LIN {X 0,Y 311.55,Z 599.519,A -85,B 0,C 180,E1 -15563.524,E2 -15563.524} C_VEL
LIN {X 0,Y 311.702,Z 601.489,A -85,B 0,C 180,E1 -15564.826,E2 -15564.826} C_VEL
LIN {X 0,Y 311.941,Z 602.986,A -85,B 0,C 180,E1 -15566.124,E2 -15566.124} C_VEL
LIN {X 0,Y 312.344,Z 604.721,A -85,B 0,C 180,E1 -15568.711,E2 -15568.711} C_VEL
LIN {X 0,Y 312.557,Z 604.974,A -85,B 0,C 180,E1 -15570,E2 -15570} C_VEL
LIN {X 0,Y 312.346,Z 604.715,A -85,B 0,C 180,E1 -15571.289,E2 -15571.289} C_VEL
LIN {X 0,Y 311.948,Z 602.974,A -85,B 0,C 180,E1 -15573.875,E2 -15573.875} C_VEL
LIN {X 0,Y 311.715,Z 601.472,A -85,B 0,C 180,E1 -15575.174,E2 -15575.174} C_VEL
LIN {X 0,Y 311.515,Z 598.688,A -85,B 0,C 180,E1 -15576.94,E2 -15576.94} C_VEL
LIN {X 0,Y 311.364,Z 594.173,A -85,B 0,C 180,E1 -15579.091,E2 -15579.091} C_VEL
LIN {X 0,Y 311.678,Z 587.813,A -85,B 0,C 180,E1 -15581.379,E2 -15581.379} C_VEL
LIN {X 0,Y 312.28,Z 580.919,A -85,B 0,C 180,E1 -15583.337,E2 -15583.337} C_VEL
LIN {X 0,Y 313.101,Z 573.765,A -85,B 0,C 180,E1 -15584.999,E2 -15584.999} C_VEL
LIN {X 0,Y 314.326,Z 565.613,A -85,B 0,C 180,E1 -15586.563,E2 -15586.563} C_VEL
LIN {X 0,Y 315.624,Z 556.565,A -85,B 0,C 180,E1 -15587.996,E2 -15587.996} C_VEL
LIN {X 0,Y 317.241,Z 545.513,A -85,B 0,C 180,E1 -15589.408,E2 -15589.408} C_VEL
LIN {X 0,Y 318.954,Z 532.942,A -85,B 0,C 180,E1 -15590.643,E2 -15590.643} C_VEL
LIN {X 0,Y 320.384,Z 520.621,A -85,B 0,C 180,E1 -15591.557,E2 -15591.557} C_VEL
LIN {X 0,Y 321.477,Z 507.646,A -85,B 0,C 180,E1 -15592.239,E2 -15592.239} C_VEL
LIN {X 0,Y 322.122,Z 493.846,A -85,B 0,C 180,E1 -15592.699,E2 -15592.699} C_VEL
LIN {X 0,Y 323.046,Z 447.747,A -85,B 0,C 180,E1 -15593.723,E2 -15593.723} C_VEL
LIN {X 0,Y 319.721,Z 414.393,A -85,B 0,C 180,E1 -15594.772,E2 -15594.772} C_VEL
LIN {X 0,Y 316.416,Z 387.78,A -85,B 0,C 180,E1 -15595.724,E2 -15595.724} C_VEL
LIN {X 0,Y 319.076,Z 366.674,A -85,B 0,C 180,E1 -15600.072,E2 -15600.072} C_VEL
LIN {X 0,Y 319.477,Z 362.665,A -85,B 0,C 180,E1 -15600.914,E2 -15600.914} C_VEL
LIN {X 0,Y 317.162,Z 351.199,A -85,B 0,C 180,E1 -15603.639,E2 -15603.639} C_VEL
LIN {X 0,Y 314.169,Z 338.968,A -85,B 0,C 180,E1 -15606.716,E2 -15606.716} C_VEL
LIN {X 0,Y 312.497,Z 332.686,A -85,B 0,C 180,E1 -15608.434,E2 -15608.434} C_VEL
LIN {X 0,Y 312.462,Z 332.564,A -85,B 0,C 180,E1 -15612.435,E2 -15612.435} C_VEL
LIN {X 0,Y 312.452,Z 332.533,A -85,B 0,C 180,E1 -15616.035,E2 -15616.035} C_VEL
LIN {X 0,Y 312.451,Z 332.552,A -85,B 0,C 180,E1 -15619.885,E2 -15619.885} C_VEL
LIN {X 0,Y 312.528,Z 332.497,A -85,B 0,C 180,E1 -15624.051,E2 -15624.051} C_VEL
LIN {X 0,Y 312.497,Z 332.555,A -85,B 0,C 180,E1 -15627.333,E2 -15627.333} C_VEL
LIN {X 0,Y 312.501,Z 332.536,A -85,B 0,C 180,E1 -15631.291,E2 -15631.291} C_VEL
LIN {X 0,Y 312.52,Z 332.555,A -85,B 0,C 180,E1 -15634.705,E2 -15634.705} C_VEL
LIN {X 0,Y 312.529,Z 332.523,A -85,B 0,C 180,E1 -15638.912,E2 -15638.912} C_VEL
LIN {X 0,Y 312.633,Z 332.53,A -85,B 0,C 180,E1 -15641.656,E2 -15641.656} C_VEL
LIN {X 0,Y 312.688,Z 332.525,A -85,B 0,C 180,E1 -15645.686,E2 -15645.686} C_VEL
LIN {X 0,Y 312.679,Z 332.535,A -85,B 0,C 180,E1 -15649.641,E2 -15649.641} C_VEL
LIN {X 0,Y 312.813,Z 332.51,A -85,B 0,C 180,E1 -15652.253,E2 -15652.253} C_VEL
LIN {X 0,Y 312.686,Z 332.523,A -85,B 0,C 180,E1 -15654.842,E2 -15654.842} C_VEL
LIN {X 0,Y 312.973,Z 332.495,A -85,B 0,C 180,E1 -15658.713,E2 -15658.713} C_VEL
LIN {X 0,Y 312.902,Z 332.502,A -85,B 0,C 180,E1 -15662.575,E2 -15662.575} C_VEL
LIN {X 0,Y 312.831,Z 332.506,A -85,B 0,C 180,E1 -15666.473,E2 -15666.473} C_VEL
LIN {X 0,Y 312.745,Z 332.515,A -85,B 0,C 180,E1 -15669.051,E2 -15669.051} C_VEL
LIN {X 0,Y 312.627,Z 332.536,A -85,B 0,C 180,E1 -15672.991,E2 -15672.991} C_VEL
LIN {X 0,Y 312.616,Z 332.531,A -85,B 0,C 180,E1 -15675.651,E2 -15675.651} C_VEL
LIN {X 0,Y 312.554,Z 332.542,A -85,B 0,C 180,E1 -15679.712,E2 -15679.712} C_VEL
LIN {X 0,Y 312.509,Z 332.553,A -85,B 0,C 180,E1 -15682.775,E2 -15682.775} C_VEL
LIN {X 0,Y 312.477,Z 332.543,A -85,B 0,C 180,E1 -15686.733,E2 -15686.733} C_VEL
LIN {X 0,Y 312.462,Z 332.51,A -85,B 0,C 180,E1 -15689.659,E2 -15689.659} C_VEL
LIN {X 0,Y 312.516,Z 332.553,A -85,B 0,C 180,E1 -15693.689,E2 -15693.689} C_VEL
LIN {X 0,Y 312.506,Z 332.535,A -85,B 0,C 180,E1 -15697.388,E2 -15697.388} C_VEL
LIN {X 0,Y 312.437,Z 332.541,A -85,B 0,C 180,E1 -15700.718,E2 -15700.718} C_VEL
LIN {X 0,Y 312.447,Z 332.562,A -85,B 0,C 180,E1 -15704.211,E2 -15704.211} C_VEL
LIN {X 0,Y 312.451,Z 332.544,A -85,B 0,C 180,E1 -15707.926,E2 -15707.926} C_VEL
LIN {X 0,Y 312.481,Z 332.544,A -85,B 0,C 180,E1 -15711.923,E2 -15711.923} C_VEL
LIN {X 0,Y 312.528,Z 332.548,A -85,B 0,C 180,E1 -15714.221,E2 -15714.221} C_VEL
LIN {X 0,Y 312.5,Z 332.545,A -85,B 0,C 180,E1 -15717.334,E2 -15717.334} C_VEL
LIN {X 0,Y 312.483,Z 332.528,A -85,B 0,C 180,E1 -15721.3,E2 -15721.3} C_VEL
LIN {X 0,Y 312.579,Z 332.675,A -85,B 0,C 180,E1 -15724.399,E2 -15724.399} C_VEL
LIN {X 0,Y 312.787,Z 333.571,A -85,B 0,C 180,E1 -15724.634,E2 -15724.634} C_VEL
LIN {X 0,Y 322.25,Z 353.976,A -85,B 0,C 180,E1 -15725.982,E2 -15725.982} C_VEL
LIN {X 0,Y 324.863,Z 359.97,A -85,B 0,C 180,E1 -15726.34,E2 -15726.34} C_VEL
LIN {X 0,Y 324.035,Z 414.568,A -85,B 0,C 180,E1 -15727.593,E2 -15727.593} C_VEL
LIN {X 0,Y 323.772,Z 427.043,A -85,B 0,C 180,E1 -15728.1,E2 -15728.1} C_VEL
LIN {X 0,Y 323.165,Z 439.993,A -85,B 0,C 180,E1 -15728.889,E2 -15728.889} C_VEL
LIN {X 0,Y 322.296,Z 452.305,A -85,B 0,C 180,E1 -15729.911,E2 -15729.911} C_VEL
LIN {X 0,Y 320.98,Z 463.869,A -85,B 0,C 180,E1 -15731.159,E2 -15731.159} C_VEL
LIN {X 0,Y 319.694,Z 474.198,A -85,B 0,C 180,E1 -15732.571,E2 -15732.571} C_VEL
LIN {X 0,Y 318.595,Z 482.613,A -85,B 0,C 180,E1 -15733.994,E2 -15733.994} C_VEL
LIN {X 0,Y 317.424,Z 490.361,A -85,B 0,C 180,E1 -15735.577,E2 -15735.577} C_VEL
LIN {X 0,Y 316.218,Z 498.029,A -85,B 0,C 180,E1 -15737.518,E2 -15737.518} C_VEL
LIN {X 0,Y 315.27,Z 503.78,A -85,B 0,C 180,E1 -15739.336,E2 -15739.336} C_VEL
LIN {X 0,Y 314.62,Z 508.048,A -85,B 0,C 180,E1 -15741.004,E2 -15741.004} C_VEL
LIN {X 0,Y 313.789,Z 511.941,A -85,B 0,C 180,E1 -15742.924,E2 -15742.924} C_VEL
LIN {X 0,Y 313.156,Z 514.815,A -85,B 0,C 180,E1 -15744.85,E2 -15744.85} C_VEL
LIN {X 0,Y 313.098,Z 516.157,A -85,B 0,C 180,E1 -15746.139,E2 -15746.139} C_VEL
LIN {X 0,Y 312.876,Z 517.135,A -85,B 0,C 180,E1 -15747.425,E2 -15747.425} C_VEL
LIN {X 0,Y 312.907,Z 517.715,A -85,B 0,C 180,E1 -15748.713,E2 -15748.713} C_VEL
LIN {X 0,Y 312.881,Z 517.941,A -85,B 0,C 180,E1 -15750,E2 -15750} C_VEL
LIN {X 0,Y 312.907,Z 517.755,A -85,B 0,C 180,E1 -15751.287,E2 -15751.287} C_VEL
LIN {X 0,Y 312.875,Z 517.201,A -85,B 0,C 180,E1 -15752.575,E2 -15752.575} C_VEL
LIN {X 0,Y 313.093,Z 516.248,A -85,B 0,C 180,E1 -15753.861,E2 -15753.861} C_VEL
LIN {X 0,Y 313.144,Z 514.948,A -85,B 0,C 180,E1 -15755.15,E2 -15755.15} C_VEL
LIN {X 0,Y 313.783,Z 512.122,A -85,B 0,C 180,E1 -15757.076,E2 -15757.076} C_VEL
LIN {X 0,Y 314.595,Z 508.294,A -85,B 0,C 180,E1 -15758.997,E2 -15758.997} C_VEL
LIN {X 0,Y 315.35,Z 503.213,A -85,B 0,C 180,E1 -15760.984,E2 -15760.984} C_VEL
LIN {X 0,Y 316.648,Z 495.971,A -85,B 0,C 180,E1 -15763.15,E2 -15763.15} C_VEL
LIN {X 0,Y 317.934,Z 487.942,A -85,B 0,C 180,E1 -15765.054,E2 -15765.054} C_VEL
LIN {X 0,Y 319.058,Z 479.718,A -85,B 0,C 180,E1 -15766.64,E2 -15766.64} C_VEL
LIN {X 0,Y 320.218,Z 470.679,A -85,B 0,C 180,E1 -15768.059,E2 -15768.059} C_VEL
LIN {X 0,Y 321.556,Z 460.163,A -85,B 0,C 180,E1 -15769.378,E2 -15769.378} C_VEL
LIN {X 0,Y 322.613,Z 448.643,A -85,B 0,C 180,E1 -15770.533,E2 -15770.533} C_VEL
LIN {X 0,Y 323.495,Z 437.366,A -85,B 0,C 180,E1 -15771.398,E2 -15771.398} C_VEL
LIN {X 0,Y 323.977,Z 425.075,A -85,B 0,C 180,E1 -15772.098,E2 -15772.098} C_VEL
LIN {X 0,Y 324.096,Z 414.763,A -85,B 0,C 180,E1 -15772.511,E2 -15772.511} C_VEL
LIN {X 0,Y 324.643,Z 374.354,A -85,B 0,C 180,E1 -15773.45,E2 -15773.45} C_VEL
LIN {X 0,Y 324.833,Z 359.99,A -85,B 0,C 180,E1 -15773.776,E2 -15773.776} C_VEL
LIN {X 0,Y 316.003,Z 340.297,A -85,B 0,C 180,E1 -15775.003,E2 -15775.003} C_VEL
LIN {X 0,Y 312.728,Z 333.371,A -85,B 0,C 180,E1 -15775.513,E2 -15775.513} C_VEL
LIN {X 0,Y 312.548,Z 332.615,A -85,B 0,C 180,E1 -15775.775,E2 -15775.775} C_VEL
LIN {X 0,Y 312.467,Z 332.547,A -85,B 0,C 180,E1 -15779.657,E2 -15779.657} C_VEL
LIN {X 0,Y 312.519,Z 332.549,A -85,B 0,C 180,E1 -15783.688,E2 -15783.688} C_VEL
LIN {X 0,Y 312.508,Z 332.537,A -85,B 0,C 180,E1 -15787.387,E2 -15787.387} C_VEL
LIN {X 0,Y 312.438,Z 332.564,A -85,B 0,C 180,E1 -15790.716,E2 -15790.716} C_VEL
LIN {X 0,Y 312.447,Z 332.543,A -85,B 0,C 180,E1 -15794.209,E2 -15794.209} C_VEL
LIN {X 0,Y 312.451,Z 332.562,A -85,B 0,C 180,E1 -15797.924,E2 -15797.924} C_VEL
LIN {X 0,Y 312.422,Z 332.551,A -85,B 0,C 180,E1 -15798.789,E2 -15798.789} C_VEL
LIN {X 0,Y 311.768,Z 332.623,A -85,B 0,C 180,E1 -15799.864,E2 -15799.864} C_VEL
LIN {X 0,Y 308.931,Z 332.977,A -85,B 0,C 180,E1 -15801.614,E2 -15801.614} C_VEL
LIN {X 0,Y 306.53,Z 333.286,A -85,B 0,C 180,E1 -15803.034,E2 -15803.034} C_VEL
LIN {X 0,Y 305.516,Z 333.423,A -85,B 0,C 180,E1 -15804.133,E2 -15804.133} C_VEL
LIN {X 0,Y 305.443,Z 333.435,A -85,B 0,C 180,E1 -15804.505,E2 -15804.505} C_VEL
LIN {X 0,Y 305.437,Z 333.407,A -85,B 0,C 180,E1 -15808.358,E2 -15808.358} C_VEL
LIN {X 0,Y 305.447,Z 333.385,A -85,B 0,C 180,E1 -15811.106,E2 -15811.106} C_VEL
LIN {X 0,Y 305.473,Z 333.423,A -85,B 0,C 180,E1 -15814.079,E2 -15814.079} C_VEL
LIN {X 0,Y 305.455,Z 333.423,A -85,B 0,C 180,E1 -15818.399,E2 -15818.399} C_VEL
LIN {X 0,Y 305.529,Z 333.427,A -85,B 0,C 180,E1 -15822.6,E2 -15822.6} C_VEL
LIN {X 0,Y 305.62,Z 333.395,A -85,B 0,C 180,E1 -15825.347,E2 -15825.347} C_VEL
LIN {X 0,Y 305.618,Z 333.413,A -85,B 0,C 180,E1 -15829.399,E2 -15829.399} C_VEL
LIN {X 0,Y 305.739,Z 333.383,A -85,B 0,C 180,E1 -15832.072,E2 -15832.072} C_VEL
LIN {X 0,Y 305.653,Z 333.412,A -85,B 0,C 180,E1 -15834.723,E2 -15834.723} C_VEL
LIN {X 0,Y 305.929,Z 333.358,A -85,B 0,C 180,E1 -15838.684,E2 -15838.684} C_VEL
LIN {X 0,Y 305.94,Z 333.371,A -85,B 0,C 180,E1 -15841.316,E2 -15841.316} C_VEL
LIN {X 0,Y 305.786,Z 333.378,A -85,B 0,C 180,E1 -15846.599,E2 -15846.599} C_VEL
LIN {X 0,Y 305.688,Z 333.405,A -85,B 0,C 180,E1 -15849.261,E2 -15849.261} C_VEL
LIN {X 0,Y 305.579,Z 333.404,A -85,B 0,C 180,E1 -15853.296,E2 -15853.296} C_VEL
LIN {X 0,Y 305.55,Z 333.425,A -85,B 0,C 180,E1 -15856.022,E2 -15856.022} C_VEL
LIN {X 0,Y 305.537,Z 333.401,A -85,B 0,C 180,E1 -15859.426,E2 -15859.426} C_VEL
LIN {X 0,Y 305.466,Z 333.427,A -85,B 0,C 180,E1 -15863.033,E2 -15863.033} C_VEL
LIN {X 0,Y 305.449,Z 333.43,A -85,B 0,C 180,E1 -15866.191,E2 -15866.191} C_VEL
LIN {X 0,Y 305.443,Z 333.417,A -85,B 0,C 180,E1 -15869.034,E2 -15869.034} C_VEL
LIN {X 0,Y 305.432,Z 333.442,A -85,B 0,C 180,E1 -15871.954,E2 -15871.954} C_VEL
LIN {X 0,Y 305.457,Z 333.421,A -85,B 0,C 180,E1 -15875.114,E2 -15875.114} C_VEL
LIN {X 0,Y 305.43,Z 333.43,A -85,B 0,C 180,E1 -15878.525,E2 -15878.525} C_VEL
LIN {X 0,Y 305.431,Z 333.432,A -85,B 0,C 180,E1 -15882.582,E2 -15882.582} C_VEL
LIN {X 0,Y 305.417,Z 333.412,A -85,B 0,C 180,E1 -15886.344,E2 -15886.344} C_VEL
LIN {X 0,Y 305.407,Z 333.418,A -85,B 0,C 180,E1 -15889.885,E2 -15889.885} C_VEL
LIN {X 0,Y 305.447,Z 333.618,A -85,B 0,C 180,E1 -15890.998,E2 -15890.998} C_VEL
LIN {X 0,Y 308.846,Z 346.507,A -85,B 0,C 180,E1 -15894.491,E2 -15894.491} C_VEL
LIN {X 0,Y 311.665,Z 358.968,A -85,B 0,C 180,E1 -15897.619,E2 -15897.619} C_VEL
LIN {X 0,Y 312.62,Z 364.164,A -85,B 0,C 180,E1 -15898.865,E2 -15898.865} C_VEL
LIN {X 0,Y 311.106,Z 375.627,A -85,B 0,C 180,E1 -15901.312,E2 -15901.312} C_VEL
LIN {X 0,Y 309.717,Z 386.706,A -85,B 0,C 180,E1 -15903.647,E2 -15903.647} C_VEL
LIN {X 0,Y 313.735,Z 419.226,A -85,B 0,C 180,E1 -15904.839,E2 -15904.839} C_VEL
LIN {X 0,Y 316.571,Z 448.811,A -85,B 0,C 180,E1 -15905.787,E2 -15905.787} C_VEL
LIN {X 0,Y 315.459,Z 497.939,A -85,B 0,C 180,E1 -15906.924,E2 -15906.924} C_VEL
LIN {X 0,Y 314.589,Z 511.17,A -85,B 0,C 180,E1 -15907.464,E2 -15907.464} C_VEL
LIN {X 0,Y 313.434,Z 523.348,A -85,B 0,C 180,E1 -15908.2,E2 -15908.2} C_VEL
LIN {X 0,Y 311.838,Z 535.654,A -85,B 0,C 180,E1 -15909.209,E2 -15909.209} C_VEL
LIN {X 0,Y 310.115,Z 547.326,A -85,B 0,C 180,E1 -15910.472,E2 -15910.472} C_VEL
LIN {X 0,Y 308.48,Z 557.874,A -85,B 0,C 180,E1 -15911.916,E2 -15911.916} C_VEL
LIN {X 0,Y 307.228,Z 566.547,A -85,B 0,C 180,E1 -15913.385,E2 -15913.385} C_VEL
LIN {X 0,Y 305.954,Z 574.893,A -85,B 0,C 180,E1 -15915.099,E2 -15915.099} C_VEL
LIN {X 0,Y 305.068,Z 582.466,A -85,B 0,C 180,E1 -15917.02,E2 -15917.02} C_VEL
LIN {X 0,Y 304.448,Z 589.797,A -85,B 0,C 180,E1 -15919.358,E2 -15919.358} C_VEL
LIN {X 0,Y 304.276,Z 594.719,A -85,B 0,C 180,E1 -15921.365,E2 -15921.365} C_VEL
LIN {X 0,Y 304.443,Z 598.525,A -85,B 0,C 180,E1 -15923.372,E2 -15923.372} C_VEL
LIN {X 0,Y 304.615,Z 600.5,A -85,B 0,C 180,E1 -15924.705,E2 -15924.705} C_VEL
LIN {X 0,Y 304.869,Z 602,A -85,B 0,C 180,E1 -15926.034,E2 -15926.034} C_VEL
LIN {X 0,Y 305.285,Z 603.738,A -85,B 0,C 180,E1 -15928.681,E2 -15928.681} C_VEL
LIN {X 0,Y 305.525,Z 603.995,A -85,B 0,C 180,E1 -15930,E2 -15930} C_VEL
LIN {X 0,Y 305.287,Z 603.732,A -85,B 0,C 180,E1 -15931.319,E2 -15931.319} C_VEL
LIN {X 0,Y 304.894,Z 601.99,A -85,B 0,C 180,E1 -15933.965,E2 -15933.965} C_VEL
LIN {X 0,Y 304.631,Z 600.482,A -85,B 0,C 180,E1 -15935.295,E2 -15935.295} C_VEL
LIN {X 0,Y 304.438,Z 597.963,A -85,B 0,C 180,E1 -15936.944,E2 -15936.944} C_VEL
LIN {X 0,Y 304.31,Z 593.178,A -85,B 0,C 180,E1 -15939.303,E2 -15939.303} C_VEL
LIN {X 0,Y 304.663,Z 586.816,A -85,B 0,C 180,E1 -15941.645,E2 -15941.645} C_VEL
LIN {X 0,Y 305.331,Z 579.923,A -85,B 0,C 180,E1 -15943.646,E2 -15943.646} C_VEL
LIN {X 0,Y 306.333,Z 572.003,A -85,B 0,C 180,E1 -15945.51,E2 -15945.51} C_VEL
LIN {X 0,Y 307.655,Z 562.765,A -85,B 0,C 180,E1 -15947.275,E2 -15947.275} C_VEL
LIN {X 0,Y 309.372,Z 552.132,A -85,B 0,C 180,E1 -15948.887,E2 -15948.887} C_VEL
LIN {X 0,Y 310.967,Z 541.643,A -85,B 0,C 180,E1 -15950.16,E2 -15950.16} C_VEL
LIN {X 0,Y 312.611,Z 530.177,A -85,B 0,C 180,E1 -15951.254,E2 -15951.254} C_VEL
LIN {X 0,Y 313.924,Z 518.382,A -85,B 0,C 180,E1 -15952.11,E2 -15952.11} C_VEL
LIN {X 0,Y 315.03,Z 504.81,A -85,B 0,C 180,E1 -15952.806,E2 -15952.806} C_VEL
LIN {X 0,Y 315.633,Z 491.252,A -85,B 0,C 180,E1 -15953.236,E2 -15953.236} C_VEL
LIN {X 0,Y 316.51,Z 448.386,A -85,B 0,C 180,E1 -15954.204,E2 -15954.204} C_VEL
LIN {X 0,Y 313.251,Z 415.354,A -85,B 0,C 180,E1 -15955.271,E2 -15955.271} C_VEL
LIN {X 0,Y 309.681,Z 387.005,A -85,B 0,C 180,E1 -15956.3,E2 -15956.3} C_VEL
LIN {X 0,Y 310.898,Z 377.146,A -85,B 0,C 180,E1 -15958.34,E2 -15958.34} C_VEL
LIN {X 0,Y 312.586,Z 364.015,A -85,B 0,C 180,E1 -15961.139,E2 -15961.139} C_VEL
LIN {X 0,Y 310.058,Z 351.698,A -85,B 0,C 180,E1 -15964.156,E2 -15964.156} C_VEL
LIN {X 0,Y 307.06,Z 339.565,A -85,B 0,C 180,E1 -15967.309,E2 -15967.309} C_VEL
LIN {X 0,Y 305.436,Z 333.537,A -85,B 0,C 180,E1 -15969.021,E2 -15969.021} C_VEL
LIN {X 0,Y 305.432,Z 333.434,A -85,B 0,C 180,E1 -15972.581,E2 -15972.581} C_VEL
LIN {X 0,Y 305.417,Z 333.413,A -85,B 0,C 180,E1 -15976.343,E2 -15976.343} C_VEL
LIN {X 0,Y 305.406,Z 333.43,A -85,B 0,C 180,E1 -15979.884,E2 -15979.884} C_VEL
LIN {X 0,Y 305.456,Z 333.372,A -85,B 0,C 180,E1 -15983.637,E2 -15983.637} C_VEL
LIN {X 0,Y 305.46,Z 333.423,A -85,B 0,C 180,E1 -15986.483,E2 -15986.483} C_VEL
LIN {X 0,Y 305.426,Z 333.432,A -85,B 0,C 180,E1 -15989.587,E2 -15989.587} C_VEL
LIN {X 0,Y 305.447,Z 333.42,A -85,B 0,C 180,E1 -15992.601,E2 -15992.601} C_VEL
LIN {X 0,Y 305.454,Z 333.438,A -85,B 0,C 180,E1 -15995.534,E2 -15995.534} C_VEL
LIN {X 0,Y 305.5,Z 333.398,A -85,B 0,C 180,E1 -15999.814,E2 -15999.814} C_VEL
LIN {X 0,Y 305.569,Z 333.419,A -85,B 0,C 180,E1 -16002.603,E2 -16002.603} C_VEL
LIN {X 0,Y 305.644,Z 333.407,A -85,B 0,C 180,E1 -16005.349,E2 -16005.349} C_VEL
LIN {X 0,Y 305.618,Z 333.412,A -85,B 0,C 180,E1 -16009.399,E2 -16009.399} C_VEL
LIN {X 0,Y 305.759,Z 333.39,A -85,B 0,C 180,E1 -16012.073,E2 -16012.073} C_VEL
LIN {X 0,Y 305.656,Z 333.398,A -85,B 0,C 180,E1 -16014.723,E2 -16014.723} C_VEL
LIN {X 0,Y 305.94,Z 333.371,A -85,B 0,C 180,E1 -16018.684,E2 -16018.684} C_VEL
LIN {X 0,Y 305.929,Z 333.357,A -85,B 0,C 180,E1 -16021.316,E2 -16021.316} C_VEL
LIN {X 0,Y 305.655,Z 333.411,A -85,B 0,C 180,E1 -16025.277,E2 -16025.277} C_VEL
LIN {X 0,Y 305.739,Z 333.382,A -85,B 0,C 180,E1 -16027.928,E2 -16027.928} C_VEL
LIN {X 0,Y 305.592,Z 333.415,A -85,B 0,C 180,E1 -16031.946,E2 -16031.946} C_VEL
LIN {X 0,Y 305.603,Z 333.398,A -85,B 0,C 180,E1 -16035.014,E2 -16035.014} C_VEL
LIN {X 0,Y 305.537,Z 333.419,A -85,B 0,C 180,E1 -16039.427,E2 -16039.427} C_VEL
LIN {X 0,Y 305.451,Z 333.433,A -85,B 0,C 180,E1 -16043.026,E2 -16043.026} C_VEL
LIN {X 0,Y 305.446,Z 333.425,A -85,B 0,C 180,E1 -16046.19,E2 -16046.19} C_VEL
LIN {X 0,Y 305.418,Z 333.388,A -85,B 0,C 180,E1 -16049.026,E2 -16049.026} C_VEL
LIN {X 0,Y 305.432,Z 333.412,A -85,B 0,C 180,E1 -16051.954,E2 -16051.954} C_VEL
LIN {X 0,Y 305.458,Z 333.437,A -85,B 0,C 180,E1 -16055.114,E2 -16055.114} C_VEL
LIN {X 0,Y 305.43,Z 333.402,A -85,B 0,C 180,E1 -16058.525,E2 -16058.525} C_VEL
LIN {X 0,Y 305.431,Z 333.437,A -85,B 0,C 180,E1 -16062.582,E2 -16062.582} C_VEL
LIN {X 0,Y 305.417,Z 333.413,A -85,B 0,C 180,E1 -16066.345,E2 -16066.345} C_VEL
LIN {X 0,Y 305.408,Z 333.443,A -85,B 0,C 180,E1 -16069.885,E2 -16069.885} C_VEL
LIN {X 0,Y 305.461,Z 333.419,A -85,B 0,C 180,E1 -16073.637,E2 -16073.637} C_VEL
LIN {X 0,Y 305.464,Z 333.426,A -85,B 0,C 180,E1 -16076.484,E2 -16076.484} C_VEL
LIN {X 0,Y 305.417,Z 333.442,A -85,B 0,C 180,E1 -16079.587,E2 -16079.587} C_VEL
LIN {X 0,Y 305.47,Z 333.433,A -85,B 0,C 180,E1 -16083.529,E2 -16083.529} C_VEL
LIN {X 0,Y 305.566,Z 333.988,A -85,B 0,C 180,E1 -16083.914,E2 -16083.914} C_VEL
LIN {X 0,Y 306.575,Z 336.366,A -85,B 0,C 180,E1 -16084.155,E2 -16084.155} C_VEL
LIN {X 0,Y 315.579,Z 355.356,A -85,B 0,C 180,E1 -16085.449,E2 -16085.449} C_VEL
LIN {X 0,Y 318.427,Z 361.87,A -85,B 0,C 180,E1 -16085.853,E2 -16085.853} C_VEL
LIN {X 0,Y 317.541,Z 414.893,A -85,B 0,C 180,E1 -16087.089,E2 -16087.089} C_VEL
LIN {X 0,Y 317.279,Z 427.5,A -85,B 0,C 180,E1 -16087.598,E2 -16087.598} C_VEL
LIN {X 0,Y 316.707,Z 439.859,A -85,B 0,C 180,E1 -16088.352,E2 -16088.352} C_VEL
LIN {X 0,Y 315.827,Z 451.578,A -85,B 0,C 180,E1 -16089.312,E2 -16089.312} C_VEL
LIN {X 0,Y 314.632,Z 462.245,A -85,B 0,C 180,E1 -16090.424,E2 -16090.424} C_VEL
LIN {X 0,Y 313.24,Z 473.086,A -85,B 0,C 180,E1 -16091.862,E2 -16091.862} C_VEL
LIN {X 0,Y 312.065,Z 481.854,A -85,B 0,C 180,E1 -16093.313,E2 -16093.313} C_VEL
LIN {X 0,Y 310.919,Z 489.88,A -85,B 0,C 180,E1 -16094.933,E2 -16094.933} C_VEL
LIN {X 0,Y 309.613,Z 497.742,A -85,B 0,C 180,E1 -16096.88,E2 -16096.88} C_VEL
LIN {X 0,Y 308.526,Z 503.652,A -85,B 0,C 180,E1 -16098.699,E2 -16098.699} C_VEL
LIN {X 0,Y 307.681,Z 509.027,A -85,B 0,C 180,E1 -16100.8,E2 -16100.8} C_VEL
LIN {X 0,Y 306.816,Z 512.92,A -85,B 0,C 180,E1 -16102.763,E2 -16102.763} C_VEL
LIN {X 0,Y 306.153,Z 515.794,A -85,B 0,C 180,E1 -16104.732,E2 -16104.732} C_VEL
LIN {X 0,Y 306.084,Z 517.136,A -85,B 0,C 180,E1 -16106.05,E2 -16106.05} C_VEL
LIN {X 0,Y 305.855,Z 518.114,A -85,B 0,C 180,E1 -16107.366,E2 -16107.366} C_VEL
LIN {X 0,Y 305.882,Z 518.693,A -85,B 0,C 180,E1 -16108.683,E2 -16108.683} C_VEL
LIN {X 0,Y 305.854,Z 518.919,A -85,B 0,C 180,E1 -16110,E2 -16110} C_VEL
LIN {X 0,Y 305.882,Z 518.732,A -85,B 0,C 180,E1 -16111.317,E2 -16111.317} C_VEL
LIN {X 0,Y 305.854,Z 518.178,A -85,B 0,C 180,E1 -16112.634,E2 -16112.634} C_VEL
LIN {X 0,Y 306.079,Z 517.226,A -85,B 0,C 180,E1 -16113.95,E2 -16113.95} C_VEL
LIN {X 0,Y 306.141,Z 515.926,A -85,B 0,C 180,E1 -16115.269,E2 -16115.269} C_VEL
LIN {X 0,Y 306.81,Z 513.099,A -85,B 0,C 180,E1 -16117.238,E2 -16117.238} C_VEL
LIN {X 0,Y 307.655,Z 509.271,A -85,B 0,C 180,E1 -16119.201,E2 -16119.201} C_VEL
LIN {X 0,Y 308.453,Z 504.189,A -85,B 0,C 180,E1 -16121.233,E2 -16121.233} C_VEL
LIN {X 0,Y 309.808,Z 496.947,A -85,B 0,C 180,E1 -16123.445,E2 -16123.445} C_VEL
LIN {X 0,Y 311.152,Z 488.917,A -85,B 0,C 180,E1 -16125.39,E2 -16125.39} C_VEL
LIN {X 0,Y 312.329,Z 480.693,A -85,B 0,C 180,E1 -16127.009,E2 -16127.009} C_VEL
LIN {X 0,Y 313.543,Z 471.653,A -85,B 0,C 180,E1 -16128.458,E2 -16128.458} C_VEL
LIN {X 0,Y 314.937,Z 461.135,A -85,B 0,C 180,E1 -16129.802,E2 -16129.802} C_VEL
LIN {X 0,Y 316.067,Z 449.459,A -85,B 0,C 180,E1 -16130.994,E2 -16130.994} C_VEL
LIN {X 0,Y 316.99,Z 437.997,A -85,B 0,C 180,E1 -16131.885,E2 -16131.885} C_VEL
LIN {X 0,Y 317.495,Z 425.422,A -85,B 0,C 180,E1 -16132.603,E2 -16132.603} C_VEL
LIN {X 0,Y 317.619,Z 415.003,A -85,B 0,C 180,E1 -16133.017,E2 -16133.017} C_VEL
LIN {X 0,Y 318.116,Z 377.17,A -85,B 0,C 180,E1 -16133.916,E2 -16133.916} C_VEL
LIN {X 0,Y 318.37,Z 361.831,A -85,B 0,C 180,E1 -16134.268,E2 -16134.268} C_VEL
LIN {X 0,Y 309.492,Z 342.166,A -85,B 0,C 180,E1 -16135.543,E2 -16135.543} C_VEL
LIN {X 0,Y 305.653,Z 334.299,A -85,B 0,C 180,E1 -16136.147,E2 -16136.147} C_VEL
LIN {X 0,Y 305.483,Z 333.487,A -85,B 0,C 180,E1 -16136.442,E2 -16136.442} C_VEL
LIN {X 0,Y 305.416,Z 333.441,A -85,B 0,C 180,E1 -16140.414,E2 -16140.414} C_VEL
LIN {X 0,Y 305.463,Z 333.432,A -85,B 0,C 180,E1 -16144.078,E2 -16144.078} C_VEL
LIN {X 0,Y 305.449,Z 333.418,A -85,B 0,C 180,E1 -16146.742,E2 -16146.742} C_VEL
LIN {X 0,Y 305.407,Z 333.441,A -85,B 0,C 180,E1 -16150.589,E2 -16150.589} C_VEL
LIN {X 0,Y 305.418,Z 333.413,A -85,B 0,C 180,E1 -16153.656,E2 -16153.656} C_VEL
LIN {X 0,Y 305.431,Z 333.438,A -85,B 0,C 180,E1 -16157.418,E2 -16157.418} C_VEL
LIN {X 0,Y 305.438,Z 333.402,A -85,B 0,C 180,E1 -16161.592,E2 -16161.592} C_VEL
LIN {X 0,Y 305.443,Z 333.435,A -85,B 0,C 180,E1 -16164.505,E2 -16164.505} C_VEL
LIN {X 0,Y 304.791,Z 333.521,A -85,B 0,C 180,E1 -16165.606,E2 -16165.606} C_VEL
LIN {X 0,Y 301.915,Z 333.864,A -85,B 0,C 180,E1 -16167.398,E2 -16167.398} C_VEL
LIN {X 0,Y 299.469,Z 334.142,A -85,B 0,C 180,E1 -16168.851,E2 -16168.851} C_VEL
LIN {X 0,Y 298.43,Z 334.257,A -85,B 0,C 180,E1 -16169.978,E2 -16169.978} C_VEL
LIN {X 0,Y 298.352,Z 334.265,A -85,B 0,C 180,E1 -16170.359,E2 -16170.359} C_VEL
LIN {X 0,Y 298.399,Z 334.298,A -85,B 0,C 180,E1 -16173.505,E2 -16173.505} C_VEL
LIN {X 0,Y 298.4,Z 334.313,A -85,B 0,C 180,E1 -16176.711,E2 -16176.711} C_VEL
LIN {X 0,Y 298.458,Z 334.303,A -85,B 0,C 180,E1 -16180.751,E2 -16180.751} C_VEL
LIN {X 0,Y 298.581,Z 334.273,A -85,B 0,C 180,E1 -16184.994,E2 -16184.994} C_VEL
LIN {X 0,Y 298.577,Z 334.291,A -85,B 0,C 180,E1 -16189.146,E2 -16189.146} C_VEL
LIN {X 0,Y 298.69,Z 334.261,A -85,B 0,C 180,E1 -16191.884,E2 -16191.884} C_VEL
LIN {X 0,Y 298.623,Z 334.286,A -85,B 0,C 180,E1 -16194.598,E2 -16194.598} C_VEL
LIN {X 0,Y 298.897,Z 334.233,A -85,B 0,C 180,E1 -16198.653,E2 -16198.653} C_VEL
LIN {X 0,Y 298.906,Z 334.247,A -85,B 0,C 180,E1 -16201.347,E2 -16201.347} C_VEL
LIN {X 0,Y 298.734,Z 334.257,A -85,B 0,C 180,E1 -16206.755,E2 -16206.755} C_VEL
LIN {X 0,Y 298.619,Z 334.285,A -85,B 0,C 180,E1 -16209.482,E2 -16209.482} C_VEL
LIN {X 0,Y 298.538,Z 334.283,A -85,B 0,C 180,E1 -16213.616,E2 -16213.616} C_VEL
LIN {X 0,Y 298.484,Z 334.305,A -85,B 0,C 180,E1 -16216.412,E2 -16216.412} C_VEL
LIN {X 0,Y 298.478,Z 334.276,A -85,B 0,C 180,E1 -16219.639,E2 -16219.639} C_VEL
LIN {X 0,Y 298.405,Z 334.309,A -85,B 0,C 180,E1 -16223.602,E2 -16223.602} C_VEL
LIN {X 0,Y 298.398,Z 334.305,A -85,B 0,C 180,E1 -16226.583,E2 -16226.583} C_VEL
LIN {X 0,Y 298.389,Z 334.302,A -85,B 0,C 180,E1 -16229.645,E2 -16229.645} C_VEL
LIN {X 0,Y 298.388,Z 334.312,A -85,B 0,C 180,E1 -16232.801,E2 -16232.801} C_VEL
LIN {X 0,Y 298.399,Z 334.308,A -85,B 0,C 180,E1 -16236.073,E2 -16236.073} C_VEL
LIN {X 0,Y 298.37,Z 334.305,A -85,B 0,C 180,E1 -16239.492,E2 -16239.492} C_VEL
LIN {X 0,Y 298.366,Z 334.298,A -85,B 0,C 180,E1 -16243.098,E2 -16243.098} C_VEL
LIN {X 0,Y 298.367,Z 334.3,A -85,B 0,C 180,E1 -16246.915,E2 -16246.915} C_VEL
LIN {X 0,Y 298.406,Z 334.505,A -85,B 0,C 180,E1 -16250.405,E2 -16250.405} C_VEL
LIN {X 0,Y 301.657,Z 346.788,A -85,B 0,C 180,E1 -16253.845,E2 -16253.845} C_VEL
LIN {X 0,Y 304.343,Z 358.541,A -85,B 0,C 180,E1 -16256.898,E2 -16256.898} C_VEL
LIN {X 0,Y 305.728,Z 365.305,A -85,B 0,C 180,E1 -16258.585,E2 -16258.585} C_VEL
LIN {X 0,Y 304.543,Z 374.638,A -85,B 0,C 180,E1 -16260.634,E2 -16260.634} C_VEL
LIN {X 0,Y 303.017,Z 385.584,A -85,B 0,C 180,E1 -16263.004,E2 -16263.004} C_VEL
LIN {X 0,Y 303.991,Z 393.267,A -85,B 0,C 180,E1 -16263.346,E2 -16263.346} C_VEL
LIN {X 0,Y 308.101,Z 427.529,A -85,B 0,C 180,E1 -16264.576,E2 -16264.576} C_VEL
LIN {X 0,Y 310.054,Z 451.277,A -85,B 0,C 180,E1 -16265.33,E2 -16265.33} C_VEL
LIN {X 0,Y 308.892,Z 496.958,A -85,B 0,C 180,E1 -16266.404,E2 -16266.404} C_VEL
LIN {X 0,Y 308.026,Z 510.189,A -85,B 0,C 180,E1 -16266.956,E2 -16266.956} C_VEL
LIN {X 0,Y 306.861,Z 522.368,A -85,B 0,C 180,E1 -16267.708,E2 -16267.708} C_VEL
LIN {X 0,Y 305.205,Z 534.67,A -85,B 0,C 180,E1 -16268.736,E2 -16268.736} C_VEL
LIN {X 0,Y 303.423,Z 546.34,A -85,B 0,C 180,E1 -16270.023,E2 -16270.023} C_VEL
LIN {X 0,Y 301.742,Z 556.89,A -85,B 0,C 180,E1 -16271.498,E2 -16271.498} C_VEL
LIN {X 0,Y 300.354,Z 565.551,A -85,B 0,C 180,E1 -16272.993,E2 -16272.993} C_VEL
LIN {X 0,Y 299.016,Z 573.577,A -85,B 0,C 180,E1 -16274.671,E2 -16274.671} C_VEL
LIN {X 0,Y 298.202,Z 580.27,A -85,B 0,C 180,E1 -16276.369,E2 -16276.369} C_VEL
LIN {X 0,Y 297.548,Z 586.912,A -85,B 0,C 180,E1 -16278.418,E2 -16278.418} C_VEL
LIN {X 0,Y 297.216,Z 592.223,A -85,B 0,C 180,E1 -16280.473,E2 -16280.473} C_VEL
LIN {X 0,Y 297.276,Z 596.397,A -85,B 0,C 180,E1 -16282.53,E2 -16282.53} C_VEL
LIN {X 0,Y 297.524,Z 599.509,A -85,B 0,C 180,E1 -16284.578,E2 -16284.578} C_VEL
LIN {X 0,Y 297.797,Z 601.013,A -85,B 0,C 180,E1 -16285.94,E2 -16285.94} C_VEL
LIN {X 0,Y 298.226,Z 602.756,A -85,B 0,C 180,E1 -16288.65,E2 -16288.65} C_VEL
LIN {X 0,Y 298.493,Z 603.016,A -85,B 0,C 180,E1 -16290,E2 -16290} C_VEL
LIN {X 0,Y 298.228,Z 602.749,A -85,B 0,C 180,E1 -16291.35,E2 -16291.35} C_VEL
LIN {X 0,Y 297.82,Z 601.003,A -85,B 0,C 180,E1 -16294.06,E2 -16294.06} C_VEL
LIN {X 0,Y 297.545,Z 599.491,A -85,B 0,C 180,E1 -16295.421,E2 -16295.421} C_VEL
LIN {X 0,Y 297.307,Z 596.369,A -85,B 0,C 180,E1 -16297.47,E2 -16297.47} C_VEL
LIN {X 0,Y 297.235,Z 592.179,A -85,B 0,C 180,E1 -16299.527,E2 -16299.527} C_VEL
LIN {X 0,Y 297.661,Z 585.819,A -85,B 0,C 180,E1 -16301.923,E2 -16301.923} C_VEL
LIN {X 0,Y 298.401,Z 578.928,A -85,B 0,C 180,E1 -16303.97,E2 -16303.97} C_VEL
LIN {X 0,Y 299.342,Z 571.721,A -85,B 0,C 180,E1 -16305.718,E2 -16305.718} C_VEL
LIN {X 0,Y 300.548,Z 563.604,A -85,B 0,C 180,E1 -16307.346,E2 -16307.346} C_VEL
LIN {X 0,Y 302.224,Z 553.481,A -85,B 0,C 180,E1 -16308.999,E2 -16308.999} C_VEL
LIN {X 0,Y 304.068,Z 542.086,A -85,B 0,C 180,E1 -16310.462,E2 -16310.462} C_VEL
LIN {X 0,Y 305.704,Z 530.956,A -85,B 0,C 180,E1 -16311.582,E2 -16311.582} C_VEL
LIN {X 0,Y 307.225,Z 518.632,A -85,B 0,C 180,E1 -16312.53,E2 -16312.53} C_VEL
LIN {X 0,Y 308.362,Z 505.646,A -85,B 0,C 180,E1 -16313.239,E2 -16313.239} C_VEL
LIN {X 0,Y 309.051,Z 491.831,A -85,B 0,C 180,E1 -16313.717,E2 -16313.717} C_VEL
LIN {X 0,Y 309.973,Z 448.754,A -85,B 0,C 180,E1 -16314.714,E2 -16314.714} C_VEL
LIN {X 0,Y 306.78,Z 415.951,A -85,B 0,C 180,E1 -16315.802,E2 -16315.802} C_VEL
LIN {X 0,Y 302.937,Z 385.854,A -85,B 0,C 180,E1 -16316.942,E2 -16316.942} C_VEL
LIN {X 0,Y 305.469,Z 368.082,A -85,B 0,C 180,E1 -16320.77,E2 -16320.77} C_VEL
LIN {X 0,Y 305.688,Z 365.239,A -85,B 0,C 180,E1 -16321.403,E2 -16321.403} C_VEL
LIN {X 0,Y 303.011,Z 352.462,A -85,B 0,C 180,E1 -16324.628,E2 -16324.628} C_VEL
LIN {X 0,Y 300.03,Z 340.575,A -85,B 0,C 180,E1 -16327.823,E2 -16327.823} C_VEL
LIN {X 0,Y 298.388,Z 334.381,A -85,B 0,C 180,E1 -16329.653,E2 -16329.653} C_VEL
LIN {X 0,Y 298.366,Z 334.3,A -85,B 0,C 180,E1 -16333.096,E2 -16333.096} C_VEL
LIN {X 0,Y 298.366,Z 334.301,A -85,B 0,C 180,E1 -16336.914,E2 -16336.914} C_VEL
LIN {X 0,Y 298.381,Z 334.271,A -85,B 0,C 180,E1 -16341.01,E2 -16341.01} C_VEL
LIN {X 0,Y 298.398,Z 334.252,A -85,B 0,C 180,E1 -16343.927,E2 -16343.927} C_VEL
LIN {X 0,Y 298.388,Z 334.312,A -85,B 0,C 180,E1 -16347.199,E2 -16347.199} C_VEL
LIN {X 0,Y 298.397,Z 334.296,A -85,B 0,C 180,E1 -16350.625,E2 -16350.625} C_VEL
LIN {X 0,Y 298.419,Z 334.312,A -85,B 0,C 180,E1 -16354.918,E2 -16354.918} C_VEL
LIN {X 0,Y 298.399,Z 334.291,A -85,B 0,C 180,E1 -16357.862,E2 -16357.862} C_VEL
LIN {X 0,Y 298.52,Z 334.277,A -85,B 0,C 180,E1 -16360.756,E2 -16360.756} C_VEL
LIN {X 0,Y 298.588,Z 334.289,A -85,B 0,C 180,E1 -16364.995,E2 -16364.995} C_VEL
LIN {X 0,Y 298.577,Z 334.288,A -85,B 0,C 180,E1 -16369.146,E2 -16369.146} C_VEL
LIN {X 0,Y 298.708,Z 334.27,A -85,B 0,C 180,E1 -16371.885,E2 -16371.885} C_VEL
LIN {X 0,Y 298.627,Z 334.272,A -85,B 0,C 180,E1 -16374.598,E2 -16374.598} C_VEL
LIN {X 0,Y 298.906,Z 334.247,A -85,B 0,C 180,E1 -16378.653,E2 -16378.653} C_VEL
LIN {X 0,Y 298.897,Z 334.233,A -85,B 0,C 180,E1 -16381.347,E2 -16381.347} C_VEL
LIN {X 0,Y 298.699,Z 334.265,A -85,B 0,C 180,E1 -16386.538,E2 -16386.538} C_VEL
LIN {X 0,Y 298.62,Z 334.277,A -85,B 0,C 180,E1 -16389.482,E2 -16389.482} C_VEL
LIN {X 0,Y 298.539,Z 334.281,A -85,B 0,C 180,E1 -16393.616,E2 -16393.616} C_VEL
LIN {X 0,Y 298.481,Z 334.3,A -85,B 0,C 180,E1 -16396.413,E2 -16396.413} C_VEL
LIN {X 0,Y 298.473,Z 334.296,A -85,B 0,C 180,E1 -16399.637,E2 -16399.637} C_VEL
LIN {X 0,Y 298.377,Z 334.319,A -85,B 0,C 180,E1 -16403.605,E2 -16403.605} C_VEL
LIN {X 0,Y 298.396,Z 334.297,A -85,B 0,C 180,E1 -16406.584,E2 -16406.584} C_VEL
LIN {X 0,Y 298.352,Z 334.265,A -85,B 0,C 180,E1 -16409.649,E2 -16409.649} C_VEL
LIN {X 0,Y 298.388,Z 334.305,A -85,B 0,C 180,E1 -16412.801,E2 -16412.801} C_VEL
LIN {X 0,Y 298.423,Z 334.297,A -85,B 0,C 180,E1 -16416.803,E2 -16416.803} C_VEL
LIN {X 0,Y 298.37,Z 334.279,A -85,B 0,C 180,E1 -16419.493,E2 -16419.493} C_VEL
LIN {X 0,Y 298.367,Z 334.32,A -85,B 0,C 180,E1 -16423.098,E2 -16423.098} C_VEL
LIN {X 0,Y 298.366,Z 334.289,A -85,B 0,C 180,E1 -16426.915,E2 -16426.915} C_VEL
LIN {X 0,Y 298.382,Z 334.31,A -85,B 0,C 180,E1 -16431.012,E2 -16431.012} C_VEL
LIN {X 0,Y 298.403,Z 334.301,A -85,B 0,C 180,E1 -16433.929,E2 -16433.929} C_VEL
LIN {X 0,Y 298.392,Z 334.302,A -85,B 0,C 180,E1 -16437.2,E2 -16437.2} C_VEL
LIN {X 0,Y 298.363,Z 334.297,A -85,B 0,C 180,E1 -16440.639,E2 -16440.639} C_VEL
LIN {X 0,Y 298.457,Z 334.438,A -85,B 0,C 180,E1 -16443.083,E2 -16443.083} C_VEL
LIN {X 0,Y 298.64,Z 335.334,A -85,B 0,C 180,E1 -16443.327,E2 -16443.327} C_VEL
LIN {X 0,Y 307.456,Z 353.436,A -85,B 0,C 180,E1 -16444.675,E2 -16444.675} C_VEL
LIN {X 0,Y 311.907,Z 363.64,A -85,B 0,C 180,E1 -16445.334,E2 -16445.334} C_VEL
LIN {X 0,Y 311.081,Z 415.287,A -85,B 0,C 180,E1 -16446.567,E2 -16446.567} C_VEL
LIN {X 0,Y 310.781,Z 428.595,A -85,B 0,C 180,E1 -16447.11,E2 -16447.11} C_VEL
LIN {X 0,Y 310.184,Z 440.845,A -85,B 0,C 180,E1 -16447.873,E2 -16447.873} C_VEL
LIN {X 0,Y 309.221,Z 453.178,A -85,B 0,C 180,E1 -16448.911,E2 -16448.911} C_VEL
LIN {X 0,Y 308.017,Z 463.228,A -85,B 0,C 180,E1 -16449.986,E2 -16449.986} C_VEL
LIN {X 0,Y 306.567,Z 474.068,A -85,B 0,C 180,E1 -16451.453,E2 -16451.453} C_VEL
LIN {X 0,Y 305.338,Z 482.835,A -85,B 0,C 180,E1 -16452.935,E2 -16452.935} C_VEL
LIN {X 0,Y 304.138,Z 490.86,A -85,B 0,C 180,E1 -16454.589,E2 -16454.589} C_VEL
LIN {X 0,Y 302.773,Z 498.722,A -85,B 0,C 180,E1 -16456.578,E2 -16456.578} C_VEL
LIN {X 0,Y 301.637,Z 504.632,A -85,B 0,C 180,E1 -16458.438,E2 -16458.438} C_VEL
LIN {X 0,Y 300.745,Z 510.006,A -85,B 0,C 180,E1 -16460.585,E2 -16460.585} C_VEL
LIN {X 0,Y 299.845,Z 513.899,A -85,B 0,C 180,E1 -16462.593,E2 -16462.593} C_VEL
LIN {X 0,Y 299.152,Z 516.773,A -85,B 0,C 180,E1 -16464.608,E2 -16464.608} C_VEL
LIN {X 0,Y 299.072,Z 518.114,A -85,B 0,C 180,E1 -16465.957,E2 -16465.957} C_VEL
LIN {X 0,Y 298.835,Z 519.092,A -85,B 0,C 180,E1 -16467.304,E2 -16467.304} C_VEL
LIN {X 0,Y 298.856,Z 519.671,A -85,B 0,C 180,E1 -16468.653,E2 -16468.653} C_VEL
LIN {X 0,Y 298.827,Z 519.897,A -85,B 0,C 180,E1 -16470,E2 -16470} C_VEL
LIN {X 0,Y 298.856,Z 519.71,A -85,B 0,C 180,E1 -16471.348,E2 -16471.348} C_VEL
LIN {X 0,Y 298.834,Z 519.156,A -85,B 0,C 180,E1 -16472.696,E2 -16472.696} C_VEL
LIN {X 0,Y 299.067,Z 518.204,A -85,B 0,C 180,E1 -16474.043,E2 -16474.043} C_VEL
LIN {X 0,Y 299.139,Z 516.904,A -85,B 0,C 180,E1 -16475.392,E2 -16475.392} C_VEL
LIN {X 0,Y 299.84,Z 514.076,A -85,B 0,C 180,E1 -16477.407,E2 -16477.407} C_VEL
LIN {X 0,Y 300.72,Z 510.247,A -85,B 0,C 180,E1 -16479.415,E2 -16479.415} C_VEL
LIN {X 0,Y 301.563,Z 505.166,A -85,B 0,C 180,E1 -16481.493,E2 -16481.493} C_VEL
LIN {X 0,Y 302.977,Z 497.923,A -85,B 0,C 180,E1 -16483.754,E2 -16483.754} C_VEL
LIN {X 0,Y 304.381,Z 489.893,A -85,B 0,C 180,E1 -16485.741,E2 -16485.741} C_VEL
LIN {X 0,Y 305.613,Z 481.668,A -85,B 0,C 180,E1 -16487.394,E2 -16487.394} C_VEL
LIN {X 0,Y 306.869,Z 472.629,A -85,B 0,C 180,E1 -16488.874,E2 -16488.874} C_VEL
LIN {X 0,Y 308.329,Z 462.111,A -85,B 0,C 180,E1 -16490.245,E2 -16490.245} C_VEL
LIN {X 0,Y 309.515,Z 450.431,A -85,B 0,C 180,E1 -16491.46,E2 -16491.46} C_VEL
LIN {X 0,Y 310.475,Z 438.967,A -85,B 0,C 180,E1 -16492.368,E2 -16492.368} C_VEL
LIN {X 0,Y 310.998,Z 426.591,A -85,B 0,C 180,E1 -16493.093,E2 -16493.093} C_VEL
LIN {X 0,Y 311.156,Z 415.265,A -85,B 0,C 180,E1 -16493.544,E2 -16493.544} C_VEL
LIN {X 0,Y 311.749,Z 375.035,A -85,B 0,C 180,E1 -16494.513,E2 -16494.513} C_VEL
LIN {X 0,Y 311.928,Z 363.716,A -85,B 0,C 180,E1 -16494.78,E2 -16494.78} C_VEL
LIN {X 0,Y 302.966,Z 343.932,A -85,B 0,C 180,E1 -16496.114,E2 -16496.114} C_VEL
LIN {X 0,Y 298.632,Z 335.353,A -85,B 0,C 180,E1 -16496.795,E2 -16496.795} C_VEL
LIN {X 0,Y 298.424,Z 334.397,A -85,B 0,C 180,E1 -16497.082,E2 -16497.082} C_VEL
LIN {X 0,Y 298.372,Z 334.316,A -85,B 0,C 180,E1 -16501.211,E2 -16501.211} C_VEL
LIN {X 0,Y 298.428,Z 334.311,A -85,B 0,C 180,E1 -16504.487,E2 -16504.487} C_VEL
LIN {X 0,Y 298.386,Z 334.296,A -85,B 0,C 180,E1 -16507.761,E2 -16507.761} C_VEL
LIN {X 0,Y 298.345,Z 334.315,A -85,B 0,C 180,E1 -16511.267,E2 -16511.267} C_VEL
LIN {X 0,Y 298.352,Z 334.307,A -85,B 0,C 180,E1 -16515.034,E2 -16515.034} C_VEL
LIN {X 0,Y 298.344,Z 334.304,A -85,B 0,C 180,E1 -16518.921,E2 -16518.921} C_VEL
LIN {X 0,Y 298.383,Z 334.287,A -85,B 0,C 180,E1 -16522.237,E2 -16522.237} C_VEL
LIN {X 0,Y 298.404,Z 334.313,A -85,B 0,C 180,E1 -16525.58,E2 -16525.58} C_VEL
LIN {X 0,Y 298.367,Z 334.279,A -85,B 0,C 180,E1 -16528.788,E2 -16528.788} C_VEL
LIN {X 0,Y 298.352,Z 334.265,A -85,B 0,C 180,E1 -16530.359,E2 -16530.359} C_VEL
LIN {X 0,Y 297.691,Z 334.355,A -85,B 0,C 180,E1 -16531.487,E2 -16531.487} C_VEL
LIN {X 0,Y 294.816,Z 334.74,A -85,B 0,C 180,E1 -16533.323,E2 -16533.323} C_VEL
LIN {X 0,Y 292.399,Z 335.059,A -85,B 0,C 180,E1 -16534.813,E2 -16534.813} C_VEL
LIN {X 0,Y 291.403,Z 335.186,A -85,B 0,C 180,E1 -16535.968,E2 -16535.968} C_VEL
LIN {X 0,Y 291.345,Z 335.194,A -85,B 0,C 180,E1 -16536.359,E2 -16536.359} C_VEL
LIN {X 0,Y 291.382,Z 335.178,A -85,B 0,C 180,E1 -16540.265,E2 -16540.265} C_VEL
LIN {X 0,Y 291.493,Z 335.158,A -85,B 0,C 180,E1 -16544.665,E2 -16544.665} C_VEL
LIN {X 0,Y 291.523,Z 335.171,A -85,B 0,C 180,E1 -16548.88,E2 -16548.88} C_VEL
LIN {X 0,Y 291.644,Z 335.139,A -85,B 0,C 180,E1 -16551.687,E2 -16551.687} C_VEL
LIN {X 0,Y 291.592,Z 335.159,A -85,B 0,C 180,E1 -16554.468,E2 -16554.468} C_VEL
LIN {X 0,Y 291.865,Z 335.109,A -85,B 0,C 180,E1 -16558.62,E2 -16558.62} C_VEL
LIN {X 0,Y 291.873,Z 335.123,A -85,B 0,C 180,E1 -16561.38,E2 -16561.38} C_VEL
LIN {X 0,Y 291.686,Z 335.135,A -85,B 0,C 180,E1 -16566.919,E2 -16566.919} C_VEL
LIN {X 0,Y 291.562,Z 335.165,A -85,B 0,C 180,E1 -16569.714,E2 -16569.714} C_VEL
LIN {X 0,Y 291.509,Z 335.16,A -85,B 0,C 180,E1 -16573.951,E2 -16573.951} C_VEL
LIN {X 0,Y 291.437,Z 335.18,A -85,B 0,C 180,E1 -16576.821,E2 -16576.821} C_VEL
LIN {X 0,Y 291.42,Z 335.152,A -85,B 0,C 180,E1 -16579.86,E2 -16579.86} C_VEL
LIN {X 0,Y 291.343,Z 335.193,A -85,B 0,C 180,E1 -16584.21,E2 -16584.21} C_VEL
LIN {X 0,Y 291.346,Z 335.176,A -85,B 0,C 180,E1 -16587.279,E2 -16587.279} C_VEL
LIN {X 0,Y 291.314,Z 335.191,A -85,B 0,C 180,E1 -16590.44,E2 -16590.44} C_VEL
LIN {X 0,Y 291.339,Z 335.181,A -85,B 0,C 180,E1 -16593.699,E2 -16593.699} C_VEL
LIN {X 0,Y 291.349,Z 335.194,A -85,B 0,C 180,E1 -16597.248,E2 -16597.248} C_VEL
LIN {X 0,Y 291.297,Z 335.195,A -85,B 0,C 180,E1 -16600.649,E2 -16600.649} C_VEL
LIN {X 0,Y 291.278,Z 335.162,A -85,B 0,C 180,E1 -16604.404,E2 -16604.404} C_VEL
LIN {X 0,Y 291.292,Z 335.195,A -85,B 0,C 180,E1 -16608.412,E2 -16608.412} C_VEL
LIN {X 0,Y 291.356,Z 335.386,A -85,B 0,C 180,E1 -16609.774,E2 -16609.774} C_VEL
LIN {X 0,Y 294.696,Z 347.923,A -85,B 0,C 180,E1 -16613.402,E2 -16613.402} C_VEL
LIN {X 0,Y 297.589,Z 360.544,A -85,B 0,C 180,E1 -16616.777,E2 -16616.777} C_VEL
LIN {X 0,Y 298.865,Z 367.474,A -85,B 0,C 180,E1 -16618.538,E2 -16618.538} C_VEL
LIN {X 0,Y 296.688,Z 381.677,A -85,B 0,C 180,E1 -16621.722,E2 -16621.722} C_VEL
LIN {X 0,Y 296.337,Z 384.913,A -85,B 0,C 180,E1 -16622.383,E2 -16622.383} C_VEL
LIN {X 0,Y 300.566,Z 418.35,A -85,B 0,C 180,E1 -16623.683,E2 -16623.683} C_VEL
LIN {X 0,Y 303.507,Z 449.322,A -85,B 0,C 180,E1 -16624.736,E2 -16624.736} C_VEL
LIN {X 0,Y 302.37,Z 496.112,A -85,B 0,C 180,E1 -16625.868,E2 -16625.868} C_VEL
LIN {X 0,Y 301.505,Z 509.233,A -85,B 0,C 180,E1 -16626.429,E2 -16626.429} C_VEL
LIN {X 0,Y 300.284,Z 521.384,A -85,B 0,C 180,E1 -16627.193,E2 -16627.193} C_VEL
LIN {X 0,Y 298.601,Z 533.686,A -85,B 0,C 180,E1 -16628.242,E2 -16628.242} C_VEL
LIN {X 0,Y 296.766,Z 545.357,A -85,B 0,C 180,E1 -16629.555,E2 -16629.555} C_VEL
LIN {X 0,Y 295.034,Z 555.907,A -85,B 0,C 180,E1 -16631.061,E2 -16631.061} C_VEL
LIN {X 0,Y 293.49,Z 564.554,A -85,B 0,C 180,E1 -16632.583,E2 -16632.583} C_VEL
LIN {X 0,Y 291.977,Z 573.388,A -85,B 0,C 180,E1 -16634.495,E2 -16634.495} C_VEL
LIN {X 0,Y 291.262,Z 579.278,A -85,B 0,C 180,E1 -16636.037,E2 -16636.037} C_VEL
LIN {X 0,Y 290.551,Z 585.919,A -85,B 0,C 180,E1 -16638.135,E2 -16638.135} C_VEL
LIN {X 0,Y 290.175,Z 591.23,A -85,B 0,C 180,E1 -16640.239,E2 -16640.239} C_VEL
LIN {X 0,Y 290.207,Z 595.405,A -85,B 0,C 180,E1 -16642.346,E2 -16642.346} C_VEL
LIN {X 0,Y 290.431,Z 598.518,A -85,B 0,C 180,E1 -16644.446,E2 -16644.446} C_VEL
LIN {X 0,Y 290.71,Z 600.025,A -85,B 0,C 180,E1 -16645.841,E2 -16645.841} C_VEL
LIN {X 0,Y 291.167,Z 601.774,A -85,B 0,C 180,E1 -16648.617,E2 -16648.617} C_VEL
LIN {X 0,Y 291.459,Z 602.038,A -85,B 0,C 180,E1 -16650,E2 -16650} C_VEL
LIN {X 0,Y 291.169,Z 601.767,A -85,B 0,C 180,E1 -16651.383,E2 -16651.383} C_VEL
LIN {X 0,Y 290.732,Z 600.013,A -85,B 0,C 180,E1 -16654.159,E2 -16654.159} C_VEL
LIN {X 0,Y 290.456,Z 598.499,A -85,B 0,C 180,E1 -16655.554,E2 -16655.554} C_VEL
LIN {X 0,Y 290.222,Z 595.374,A -85,B 0,C 180,E1 -16657.653,E2 -16657.653} C_VEL
LIN {X 0,Y 290.187,Z 591.183,A -85,B 0,C 180,E1 -16659.76,E2 -16659.76} C_VEL
LIN {X 0,Y 290.641,Z 584.818,A -85,B 0,C 180,E1 -16662.215,E2 -16662.215} C_VEL
LIN {X 0,Y 291.483,Z 577.933,A -85,B 0,C 180,E1 -16664.308,E2 -16664.308} C_VEL
LIN {X 0,Y 292.501,Z 570.642,A -85,B 0,C 180,E1 -16666.115,E2 -16666.115} C_VEL
LIN {X 0,Y 294.028,Z 560.769,A -85,B 0,C 180,E1 -16668.103,E2 -16668.103} C_VEL
LIN {X 0,Y 295.919,Z 550.141,A -85,B 0,C 180,E1 -16669.781,E2 -16669.781} C_VEL
LIN {X 0,Y 297.839,Z 538.207,A -85,B 0,C 180,E1 -16671.272,E2 -16671.272} C_VEL
LIN {X 0,Y 299.668,Z 526.235,A -85,B 0,C 180,E1 -16672.402,E2 -16672.402} C_VEL
LIN {X 0,Y 301.053,Z 513.774,A -85,B 0,C 180,E1 -16673.29,E2 -16673.29} C_VEL
LIN {X 0,Y 302.026,Z 501.255,A -85,B 0,C 180,E1 -16673.924,E2 -16673.924} C_VEL
LIN {X 0,Y 302.593,Z 488.404,A -85,B 0,C 180,E1 -16674.322,E2 -16674.322} C_VEL
LIN {X 0,Y 303.473,Z 449.439,A -85,B 0,C 180,E1 -16675.237,E2 -16675.237} C_VEL
LIN {X 0,Y 300.398,Z 417.201,A -85,B 0,C 180,E1 -16676.333,E2 -16676.333} C_VEL
LIN {X 0,Y 296.551,Z 387.18,A -85,B 0,C 180,E1 -16677.479,E2 -16677.479} C_VEL
LIN {X 0,Y 296.265,Z 384.493,A -85,B 0,C 180,E1 -16677.648,E2 -16677.648} C_VEL
LIN {X 0,Y 298.683,Z 368.631,A -85,B 0,C 180,E1 -16681.175,E2 -16681.175} C_VEL
LIN {X 0,Y 298.706,Z 366.062,A -85,B 0,C 180,E1 -16681.777,E2 -16681.777} C_VEL
LIN {X 0,Y 296.007,Z 353.38,A -85,B 0,C 180,E1 -16685.076,E2 -16685.076} C_VEL
LIN {X 0,Y 293.002,Z 341.441,A -85,B 0,C 180,E1 -16688.401,E2 -16688.401} C_VEL
LIN {X 0,Y 291.342,Z 335.288,A -85,B 0,C 180,E1 -16690.243,E2 -16690.243} C_VEL
LIN {X 0,Y 291.278,Z 335.164,A -85,B 0,C 180,E1 -16694.403,E2 -16694.403} C_VEL
LIN {X 0,Y 291.291,Z 335.203,A -85,B 0,C 180,E1 -16698.411,E2 -16698.411} C_VEL
LIN {X 0,Y 291.328,Z 335.145,A -85,B 0,C 180,E1 -16701.154,E2 -16701.154} C_VEL
LIN {X 0,Y 291.35,Z 335.139,A -85,B 0,C 180,E1 -16704.624,E2 -16704.624} C_VEL
LIN {X 0,Y 291.361,Z 335.193,A -85,B 0,C 180,E1 -16707.949,E2 -16707.949} C_VEL
LIN {X 0,Y 291.338,Z 335.171,A -85,B 0,C 180,E1 -16711.154,E2 -16711.154} C_VEL
LIN {X 0,Y 291.344,Z 335.194,A -85,B 0,C 180,E1 -16714.265,E2 -16714.265} C_VEL
LIN {X 0,Y 291.356,Z 335.176,A -85,B 0,C 180,E1 -16717.297,E2 -16717.297} C_VEL
LIN {X 0,Y 291.454,Z 335.15,A -85,B 0,C 180,E1 -16720.27,E2 -16720.27} C_VEL
LIN {X 0,Y 291.536,Z 335.167,A -85,B 0,C 180,E1 -16724.634,E2 -16724.634} C_VEL
LIN {X 0,Y 291.523,Z 335.166,A -85,B 0,C 180,E1 -16728.88,E2 -16728.88} C_VEL
LIN {X 0,Y 291.659,Z 335.15,A -85,B 0,C 180,E1 -16731.687,E2 -16731.687} C_VEL
LIN {X 0,Y 291.597,Z 335.146,A -85,B 0,C 180,E1 -16734.468,E2 -16734.468} C_VEL
LIN {X 0,Y 291.873,Z 335.123,A -85,B 0,C 180,E1 -16738.62,E2 -16738.62} C_VEL
LIN {X 0,Y 291.865,Z 335.109,A -85,B 0,C 180,E1 -16741.38,E2 -16741.38} C_VEL
LIN {X 0,Y 291.679,Z 335.137,A -85,B 0,C 180,E1 -16746.92,E2 -16746.92} C_VEL
LIN {X 0,Y 291.563,Z 335.158,A -85,B 0,C 180,E1 -16749.714,E2 -16749.714} C_VEL
LIN {X 0,Y 291.509,Z 335.154,A -85,B 0,C 180,E1 -16753.951,E2 -16753.951} C_VEL
LIN {X 0,Y 291.435,Z 335.178,A -85,B 0,C 180,E1 -16756.821,E2 -16756.821} C_VEL
LIN {X 0,Y 291.42,Z 335.172,A -85,B 0,C 180,E1 -16759.86,E2 -16759.86} C_VEL
LIN {X 0,Y 291.321,Z 335.196,A -85,B 0,C 180,E1 -16764.212,E2 -16764.212} C_VEL
LIN {X 0,Y 291.323,Z 335.165,A -85,B 0,C 180,E1 -16767.282,E2 -16767.282} C_VEL
LIN {X 0,Y 291.297,Z 335.147,A -85,B 0,C 180,E1 -16770.442,E2 -16770.442} C_VEL
LIN {X 0,Y 291.34,Z 335.19,A -85,B 0,C 180,E1 -16773.699,E2 -16773.699} C_VEL
LIN {X 0,Y 291.349,Z 335.17,A -85,B 0,C 180,E1 -16777.248,E2 -16777.248} C_VEL
LIN {X 0,Y 291.296,Z 335.17,A -85,B 0,C 180,E1 -16780.649,E2 -16780.649} C_VEL
LIN {X 0,Y 291.28,Z 335.199,A -85,B 0,C 180,E1 -16784.404,E2 -16784.404} C_VEL
LIN {X 0,Y 291.292,Z 335.184,A -85,B 0,C 180,E1 -16788.412,E2 -16788.412} C_VEL
LIN {X 0,Y 291.332,Z 335.186,A -85,B 0,C 180,E1 -16791.156,E2 -16791.156} C_VEL
LIN {X 0,Y 291.354,Z 335.191,A -85,B 0,C 180,E1 -16794.626,E2 -16794.626} C_VEL
LIN {X 0,Y 291.365,Z 335.178,A -85,B 0,C 180,E1 -16797.951,E2 -16797.951} C_VEL
LIN {X 0,Y 291.378,Z 335.338,A -85,B 0,C 180,E1 -16802.375,E2 -16802.375} C_VEL
LIN {X 0,Y 291.585,Z 336.214,A -85,B 0,C 180,E1 -16802.622,E2 -16802.622} C_VEL
LIN {X 0,Y 300.65,Z 354.542,A -85,B 0,C 180,E1 -16804.06,E2 -16804.06} C_VEL
LIN {X 0,Y 305.477,Z 365.486,A -85,B 0,C 180,E1 -16804.8,E2 -16804.8} C_VEL
LIN {X 0,Y 304.645,Z 415.73,A -85,B 0,C 180,E1 -16806.025,E2 -16806.025} C_VEL
LIN {X 0,Y 304.335,Z 429.076,A -85,B 0,C 180,E1 -16806.567,E2 -16806.567} C_VEL
LIN {X 0,Y 303.685,Z 441.831,A -85,B 0,C 180,E1 -16807.373,E2 -16807.373} C_VEL
LIN {X 0,Y 302.718,Z 453.546,A -85,B 0,C 180,E1 -16808.373,E2 -16808.373} C_VEL
LIN {X 0,Y 301.421,Z 464.211,A -85,B 0,C 180,E1 -16809.529,E2 -16809.529} C_VEL
LIN {X 0,Y 299.91,Z 475.049,A -85,B 0,C 180,E1 -16811.026,E2 -16811.026} C_VEL
LIN {X 0,Y 298.625,Z 483.816,A -85,B 0,C 180,E1 -16812.539,E2 -16812.539} C_VEL
LIN {X 0,Y 297.368,Z 491.841,A -85,B 0,C 180,E1 -16814.229,E2 -16814.229} C_VEL
LIN {X 0,Y 295.941,Z 499.702,A -85,B 0,C 180,E1 -16816.262,E2 -16816.262} C_VEL
LIN {X 0,Y 294.755,Z 505.612,A -85,B 0,C 180,E1 -16818.164,E2 -16818.164} C_VEL
LIN {X 0,Y 293.814,Z 510.986,A -85,B 0,C 180,E1 -16820.361,E2 -16820.361} C_VEL
LIN {X 0,Y 292.878,Z 514.877,A -85,B 0,C 180,E1 -16822.416,E2 -16822.416} C_VEL
LIN {X 0,Y 292.152,Z 517.753,A -85,B 0,C 180,E1 -16824.478,E2 -16824.478} C_VEL
LIN {X 0,Y 292.06,Z 519.093,A -85,B 0,C 180,E1 -16825.86,E2 -16825.86} C_VEL
LIN {X 0,Y 291.815,Z 520.07,A -85,B 0,C 180,E1 -16827.239,E2 -16827.239} C_VEL
LIN {X 0,Y 291.831,Z 520.649,A -85,B 0,C 180,E1 -16828.62,E2 -16828.62} C_VEL
LIN {X 0,Y 291.8,Z 520.875,A -85,B 0,C 180,E1 -16830,E2 -16830} C_VEL
LIN {X 0,Y 291.831,Z 520.688,A -85,B 0,C 180,E1 -16831.38,E2 -16831.38} C_VEL
LIN {X 0,Y 291.814,Z 520.133,A -85,B 0,C 180,E1 -16832.761,E2 -16832.761} C_VEL
LIN {X 0,Y 292.055,Z 519.181,A -85,B 0,C 180,E1 -16834.14,E2 -16834.14} C_VEL
LIN {X 0,Y 292.139,Z 517.882,A -85,B 0,C 180,E1 -16835.522,E2 -16835.522} C_VEL
LIN {X 0,Y 292.872,Z 515.053,A -85,B 0,C 180,E1 -16837.584,E2 -16837.584} C_VEL
LIN {X 0,Y 293.789,Z 511.224,A -85,B 0,C 180,E1 -16839.64,E2 -16839.64} C_VEL
LIN {X 0,Y 294.679,Z 506.142,A -85,B 0,C 180,E1 -16841.765,E2 -16841.765} C_VEL
LIN {X 0,Y 296.156,Z 498.899,A -85,B 0,C 180,E1 -16844.078,E2 -16844.078} C_VEL
LIN {X 0,Y 297.622,Z 490.869,A -85,B 0,C 180,E1 -16846.109,E2 -16846.109} C_VEL
LIN {X 0,Y 298.911,Z 482.643,A -85,B 0,C 180,E1 -16847.797,E2 -16847.797} C_VEL
LIN {X 0,Y 300.206,Z 473.607,A -85,B 0,C 180,E1 -16849.309,E2 -16849.309} C_VEL
LIN {X 0,Y 301.902,Z 462.058,A -85,B 0,C 180,E1 -16850.825,E2 -16850.825} C_VEL
LIN {X 0,Y 303.084,Z 450.443,A -85,B 0,C 180,E1 -16852.037,E2 -16852.037} C_VEL
LIN {X 0,Y 304.055,Z 438.686,A -85,B 0,C 180,E1 -16852.957,E2 -16852.957} C_VEL
LIN {X 0,Y 304.579,Z 426.209,A -85,B 0,C 180,E1 -16853.676,E2 -16853.676} C_VEL
LIN {X 0,Y 304.727,Z 415.603,A -85,B 0,C 180,E1 -16854.091,E2 -16854.091} C_VEL
LIN {X 0,Y 305.319,Z 377.229,A -85,B 0,C 180,E1 -16855.032,E2 -16855.032} C_VEL
LIN {X 0,Y 305.514,Z 365.564,A -85,B 0,C 180,E1 -16855.314,E2 -16855.314} C_VEL
LIN {X 0,Y 297.199,Z 347.235,A -85,B 0,C 180,E1 -16856.596,E2 -16856.596} C_VEL
LIN {X 0,Y 291.595,Z 336.217,A -85,B 0,C 180,E1 -16857.501,E2 -16857.501} C_VEL
LIN {X 0,Y 291.382,Z 335.244,A -85,B 0,C 180,E1 -16857.811,E2 -16857.811} C_VEL
LIN {X 0,Y 291.365,Z 335.178,A -85,B 0,C 180,E1 -16862.05,E2 -16862.05} C_VEL
LIN {X 0,Y 291.353,Z 335.192,A -85,B 0,C 180,E1 -16865.374,E2 -16865.374} C_VEL
LIN {X 0,Y 291.304,Z 335.188,A -85,B 0,C 180,E1 -16868.849,E2 -16868.849} C_VEL
LIN {X 0,Y 291.284,Z 335.175,A -85,B 0,C 180,E1 -16872.498,E2 -16872.498} C_VEL
LIN {X 0,Y 291.286,Z 335.202,A -85,B 0,C 180,E1 -16876.37,E2 -16876.37} C_VEL
LIN {X 0,Y 291.353,Z 335.152,A -85,B 0,C 180,E1 -16880.524,E2 -16880.524} C_VEL
LIN {X 0,Y 291.382,Z 335.167,A -85,B 0,C 180,E1 -16882.916,E2 -16882.916} C_VEL
LIN {X 0,Y 291.34,Z 335.191,A -85,B 0,C 180,E1 -16886.301,E2 -16886.301} C_VEL
LIN {X 0,Y 291.33,Z 335.139,A -85,B 0,C 180,E1 -16890.278,E2 -16890.278} C_VEL
LIN {X 0,Y 291.337,Z 335.185,A -85,B 0,C 180,E1 -16894.264,E2 -16894.264} C_VEL
LIN {X 0,Y 291.345,Z 335.194,A -85,B 0,C 180,E1 -16896.359,E2 -16896.359} C_VEL
LIN {X 0,Y 290.725,Z 335.275,A -85,B 0,C 180,E1 -16897.513,E2 -16897.513} C_VEL
LIN {X 0,Y 287.852,Z 335.629,A -85,B 0,C 180,E1 -16899.391,E2 -16899.391} C_VEL
LIN {X 0,Y 285.41,Z 335.93,A -85,B 0,C 180,E1 -16900.917,E2 -16900.917} C_VEL
LIN {X 0,Y 284.402,Z 336.059,A -85,B 0,C 180,E1 -16902.1,E2 -16902.1} C_VEL
LIN {X 0,Y 284.344,Z 336.063,A -85,B 0,C 180,E1 -16902.501,E2 -16902.501} C_VEL
LIN {X 0,Y 284.458,Z 336.031,A -85,B 0,C 180,E1 -16905.696,E2 -16905.696} C_VEL
LIN {X 0,Y 284.509,Z 336.041,A -85,B 0,C 180,E1 -16910.043,E2 -16910.043} C_VEL
LIN {X 0,Y 284.634,Z 336.013,A -85,B 0,C 180,E1 -16912.908,E2 -16912.908} C_VEL
LIN {X 0,Y 284.832,Z 335.985,A -85,B 0,C 180,E1 -16918.586,E2 -16918.586} C_VEL
LIN {X 0,Y 284.839,Z 335.999,A -85,B 0,C 180,E1 -16921.414,E2 -16921.414} C_VEL
LIN {X 0,Y 284.641,Z 336.014,A -85,B 0,C 180,E1 -16927.091,E2 -16927.091} C_VEL
LIN {X 0,Y 284.508,Z 336.046,A -85,B 0,C 180,E1 -16929.957,E2 -16929.957} C_VEL
LIN {X 0,Y 284.458,Z 336.041,A -85,B 0,C 180,E1 -16934.304,E2 -16934.304} C_VEL
LIN {X 0,Y 284.37,Z 336.045,A -85,B 0,C 180,E1 -16938.741,E2 -16938.741} C_VEL
LIN {X 0,Y 284.302,Z 336.042,A -85,B 0,C 180,E1 -16941.765,E2 -16941.765} C_VEL
LIN {X 0,Y 284.291,Z 336.072,A -85,B 0,C 180,E1 -16944.851,E2 -16944.851} C_VEL
LIN {X 0,Y 284.277,Z 336.05,A -85,B 0,C 180,E1 -16948.016,E2 -16948.016} C_VEL
LIN {X 0,Y 284.281,Z 336.073,A -85,B 0,C 180,E1 -16951.276,E2 -16951.276} C_VEL
LIN {X 0,Y 284.332,Z 336.053,A -85,B 0,C 180,E1 -16955.347,E2 -16955.347} C_VEL
LIN {X 0,Y 284.291,Z 336.066,A -85,B 0,C 180,E1 -16958.172,E2 -16958.172} C_VEL
LIN {X 0,Y 284.233,Z 336.076,A -85,B 0,C 180,E1 -16962.117,E2 -16962.117} C_VEL
LIN {X 0,Y 284.234,Z 336.045,A -85,B 0,C 180,E1 -16966.186,E2 -16966.186} C_VEL
LIN {X 0,Y 284.316,Z 336.307,A -85,B 0,C 180,E1 -16969.12,E2 -16969.12} C_VEL
LIN {X 0,Y 287.535,Z 348.362,A -85,B 0,C 180,E1 -16972.732,E2 -16972.732} C_VEL
LIN {X 0,Y 290.172,Z 359.441,A -85,B 0,C 180,E1 -16975.822,E2 -16975.822} C_VEL
LIN {X 0,Y 291.845,Z 367.703,A -85,B 0,C 180,E1 -16978.01,E2 -16978.01} C_VEL
LIN {X 0,Y 291.688,Z 371.004,A -85,B 0,C 180,E1 -16978.801,E2 -16978.801} C_VEL
LIN {X 0,Y 289.683,Z 383.632,A -85,B 0,C 180,E1 -16981.666,E2 -16981.666} C_VEL
LIN {X 0,Y 292.4,Z 404.152,A -85,B 0,C 180,E1 -16982.541,E2 -16982.541} C_VEL
LIN {X 0,Y 296.186,Z 439.086,A -85,B 0,C 180,E1 -16983.826,E2 -16983.826} C_VEL
LIN {X 0,Y 297.11,Z 452.191,A -85,B 0,C 180,E1 -16984.252,E2 -16984.252} C_VEL
LIN {X 0,Y 295.905,Z 494.742,A -85,B 0,C 180,E1 -16985.29,E2 -16985.29} C_VEL
LIN {X 0,Y 294.972,Z 508.375,A -85,B 0,C 180,E1 -16985.882,E2 -16985.882} C_VEL
LIN {X 0,Y 293.602,Z 521.522,A -85,B 0,C 180,E1 -16986.737,E2 -16986.737} C_VEL
LIN {X 0,Y 292.005,Z 532.701,A -85,B 0,C 180,E1 -16987.724,E2 -16987.724} C_VEL
LIN {X 0,Y 290.073,Z 544.365,A -85,B 0,C 180,E1 -16989.062,E2 -16989.062} C_VEL
LIN {X 0,Y 288.269,Z 554.914,A -85,B 0,C 180,E1 -16990.599,E2 -16990.599} C_VEL
LIN {X 0,Y 286.642,Z 563.556,A -85,B 0,C 180,E1 -16992.153,E2 -16992.153} C_VEL
LIN {X 0,Y 285.219,Z 571.726,A -85,B 0,C 180,E1 -16993.944,E2 -16993.944} C_VEL
LIN {X 0,Y 284.13,Z 579.475,A -85,B 0,C 180,E1 -16996.045,E2 -16996.045} C_VEL
LIN {X 0,Y 283.334,Z 586.808,A -85,B 0,C 180,E1 -16998.555,E2 -16998.555} C_VEL
LIN {X 0,Y 283.071,Z 591.735,A -85,B 0,C 180,E1 -17000.713,E2 -17000.713} C_VEL
LIN {X 0,Y 283.213,Z 595.801,A -85,B 0,C 180,E1 -17003.032,E2 -17003.032} C_VEL
LIN {X 0,Y 283.626,Z 599.037,A -85,B 0,C 180,E1 -17005.737,E2 -17005.737} C_VEL
LIN {X 0,Y 284.108,Z 600.791,A -85,B 0,C 180,E1 -17008.583,E2 -17008.583} C_VEL
LIN {X 0,Y 284.425,Z 601.059,A -85,B 0,C 180,E1 -17010,E2 -17010} C_VEL
LIN {X 0,Y 284.111,Z 600.784,A -85,B 0,C 180,E1 -17011.417,E2 -17011.417} C_VEL
LIN {X 0,Y 283.646,Z 599.024,A -85,B 0,C 180,E1 -17014.263,E2 -17014.263} C_VEL
LIN {X 0,Y 283.368,Z 597.508,A -85,B 0,C 180,E1 -17015.693,E2 -17015.693} C_VEL
LIN {X 0,Y 283.121,Z 594.375,A -85,B 0,C 180,E1 -17017.847,E2 -17017.847} C_VEL
LIN {X 0,Y 283.127,Z 590.185,A -85,B 0,C 180,E1 -17020.006,E2 -17020.006} C_VEL
LIN {X 0,Y 283.647,Z 583.821,A -85,B 0,C 180,E1 -17022.521,E2 -17022.521} C_VEL
LIN {X 0,Y 284.559,Z 576.936,A -85,B 0,C 180,E1 -17024.664,E2 -17024.664} C_VEL
LIN {X 0,Y 285.524,Z 570.266,A -85,B 0,C 180,E1 -17026.369,E2 -17026.369} C_VEL
LIN {X 0,Y 286.921,Z 561.607,A -85,B 0,C 180,E1 -17028.198,E2 -17028.198} C_VEL
LIN {X 0,Y 288.809,Z 551.495,A -85,B 0,C 180,E1 -17029.918,E2 -17029.918} C_VEL
LIN {X 0,Y 290.772,Z 540.096,A -85,B 0,C 180,E1 -17031.442,E2 -17031.442} C_VEL
LIN {X 0,Y 292.547,Z 528.969,A -85,B 0,C 180,E1 -17032.605,E2 -17032.605} C_VEL
LIN {X 0,Y 294.153,Z 516.641,A -85,B 0,C 180,E1 -17033.59,E2 -17033.59} C_VEL
LIN {X 0,Y 295.326,Z 503.285,A -85,B 0,C 180,E1 -17034.348,E2 -17034.348} C_VEL
LIN {X 0,Y 296.039,Z 490.247,A -85,B 0,C 180,E1 -17034.814,E2 -17034.814} C_VEL
LIN {X 0,Y 297.043,Z 450.476,A -85,B 0,C 180,E1 -17035.769,E2 -17035.769} C_VEL
LIN {X 0,Y 294.092,Z 418.927,A -85,B 0,C 180,E1 -17036.87,E2 -17036.87} C_VEL
LIN {X 0,Y 290.311,Z 388.902,A -85,B 0,C 180,E1 -17038.047,E2 -17038.047} C_VEL
LIN {X 0,Y 289.664,Z 383.696,A -85,B 0,C 180,E1 -17038.295,E2 -17038.295} C_VEL
LIN {X 0,Y 291.894,Z 369.248,A -85,B 0,C 180,E1 -17041.579,E2 -17041.579} C_VEL
LIN {X 0,Y 291.485,Z 365.828,A -85,B 0,C 180,E1 -17042.447,E2 -17042.447} C_VEL
LIN {X 0,Y 288.842,Z 353.655,A -85,B 0,C 180,E1 -17045.729,E2 -17045.729} C_VEL
LIN {X 0,Y 285.782,Z 341.575,A -85,B 0,C 180,E1 -17049.227,E2 -17049.227} C_VEL
LIN {X 0,Y 284.296,Z 336.144,A -85,B 0,C 180,E1 -17050.939,E2 -17050.939} C_VEL
LIN {X 0,Y 284.23,Z 336.043,A -85,B 0,C 180,E1 -17054.187,E2 -17054.187} C_VEL
LIN {X 0,Y 284.236,Z 336.081,A -85,B 0,C 180,E1 -17058.118,E2 -17058.118} C_VEL
LIN {X 0,Y 284.289,Z 336.009,A -85,B 0,C 180,E1 -17061.827,E2 -17061.827} C_VEL
LIN {X 0,Y 284.303,Z 336.031,A -85,B 0,C 180,E1 -17065.35,E2 -17065.35} C_VEL
LIN {X 0,Y 284.281,Z 336.073,A -85,B 0,C 180,E1 -17068.724,E2 -17068.724} C_VEL
LIN {X 0,Y 284.277,Z 336.05,A -85,B 0,C 180,E1 -17071.984,E2 -17071.984} C_VEL
LIN {X 0,Y 284.306,Z 336.066,A -85,B 0,C 180,E1 -17076.151,E2 -17076.151} C_VEL
LIN {X 0,Y 284.383,Z 336.027,A -85,B 0,C 180,E1 -17079.898,E2 -17079.898} C_VEL
LIN {X 0,Y 284.474,Z 336.047,A -85,B 0,C 180,E1 -17084.469,E2 -17084.469} C_VEL
LIN {X 0,Y 284.477,Z 336.043,A -85,B 0,C 180,E1 -17088.601,E2 -17088.601} C_VEL
LIN {X 0,Y 284.614,Z 336.03,A -85,B 0,C 180,E1 -17091.48,E2 -17091.48} C_VEL
LIN {X 0,Y 284.567,Z 336.02,A -85,B 0,C 180,E1 -17094.331,E2 -17094.331} C_VEL
LIN {X 0,Y 284.839,Z 336,A -85,B 0,C 180,E1 -17098.586,E2 -17098.586} C_VEL
LIN {X 0,Y 284.832,Z 335.985,A -85,B 0,C 180,E1 -17101.414,E2 -17101.414} C_VEL
LIN {X 0,Y 284.635,Z 336.012,A -85,B 0,C 180,E1 -17107.092,E2 -17107.092} C_VEL
LIN {X 0,Y 284.509,Z 336.04,A -85,B 0,C 180,E1 -17109.957,E2 -17109.957} C_VEL
LIN {X 0,Y 284.458,Z 336.03,A -85,B 0,C 180,E1 -17114.304,E2 -17114.304} C_VEL
LIN {X 0,Y 284.37,Z 336.06,A -85,B 0,C 180,E1 -17118.741,E2 -17118.741} C_VEL
LIN {X 0,Y 284.298,Z 336.058,A -85,B 0,C 180,E1 -17121.766,E2 -17121.766} C_VEL
LIN {X 0,Y 284.278,Z 336.073,A -85,B 0,C 180,E1 -17124.852,E2 -17124.852} C_VEL
LIN {X 0,Y 284.255,Z 336.032,A -85,B 0,C 180,E1 -17128.019,E2 -17128.019} C_VEL
LIN {X 0,Y 284.273,Z 336.032,A -85,B 0,C 180,E1 -17131.277,E2 -17131.277} C_VEL
LIN {X 0,Y 284.333,Z 336.067,A -85,B 0,C 180,E1 -17135.347,E2 -17135.347} C_VEL
LIN {X 0,Y 284.292,Z 336.036,A -85,B 0,C 180,E1 -17138.172,E2 -17138.172} C_VEL
LIN {X 0,Y 284.234,Z 336.073,A -85,B 0,C 180,E1 -17142.118,E2 -17142.118} C_VEL
LIN {X 0,Y 284.234,Z 336.051,A -85,B 0,C 180,E1 -17146.186,E2 -17146.186} C_VEL
LIN {X 0,Y 284.281,Z 336.074,A -85,B 0,C 180,E1 -17150.03,E2 -17150.03} C_VEL
LIN {X 0,Y 284.319,Z 336.051,A -85,B 0,C 180,E1 -17153.613,E2 -17153.613} C_VEL
LIN {X 0,Y 284.305,Z 336.055,A -85,B 0,C 180,E1 -17157.191,E2 -17157.191} C_VEL
LIN {X 0,Y 284.325,Z 336.188,A -85,B 0,C 180,E1 -17161.588,E2 -17161.588} C_VEL
LIN {X 0,Y 284.578,Z 337.183,A -85,B 0,C 180,E1 -17161.888,E2 -17161.888} C_VEL
LIN {X 0,Y 294.03,Z 356,A -85,B 0,C 180,E1 -17163.442,E2 -17163.442} C_VEL
LIN {X 0,Y 299.081,Z 367.39,A -85,B 0,C 180,E1 -17164.246,E2 -17164.246} C_VEL
LIN {X 0,Y 298.23,Z 416.274,A -85,B 0,C 180,E1 -17165.461,E2 -17165.461} C_VEL
LIN {X 0,Y 297.915,Z 429.554,A -85,B 0,C 180,E1 -17166.003,E2 -17166.003} C_VEL
LIN {X 0,Y 297.289,Z 441.7,A -85,B 0,C 180,E1 -17166.766,E2 -17166.766} C_VEL
LIN {X 0,Y 296.196,Z 454.53,A -85,B 0,C 180,E1 -17167.871,E2 -17167.871} C_VEL
LIN {X 0,Y 294.851,Z 465.194,A -85,B 0,C 180,E1 -17169.051,E2 -17169.051} C_VEL
LIN {X 0,Y 293.27,Z 476.031,A -85,B 0,C 180,E1 -17170.58,E2 -17170.58} C_VEL
LIN {X 0,Y 291.927,Z 484.797,A -85,B 0,C 180,E1 -17172.125,E2 -17172.125} C_VEL
LIN {X 0,Y 290.61,Z 492.821,A -85,B 0,C 180,E1 -17173.853,E2 -17173.853} C_VEL
LIN {X 0,Y 289.119,Z 500.682,A -85,B 0,C 180,E1 -17175.932,E2 -17175.932} C_VEL
LIN {X 0,Y 287.88,Z 506.591,A -85,B 0,C 180,E1 -17177.877,E2 -17177.877} C_VEL
LIN {X 0,Y 286.888,Z 511.965,A -85,B 0,C 180,E1 -17180.126,E2 -17180.126} C_VEL
LIN {X 0,Y 285.913,Z 515.856,A -85,B 0,C 180,E1 -17182.23,E2 -17182.23} C_VEL
LIN {X 0,Y 285.153,Z 518.732,A -85,B 0,C 180,E1 -17184.342,E2 -17184.342} C_VEL
LIN {X 0,Y 285.049,Z 520.072,A -85,B 0,C 180,E1 -17185.758,E2 -17185.758} C_VEL
LIN {X 0,Y 284.795,Z 521.049,A -85,B 0,C 180,E1 -17187.171,E2 -17187.171} C_VEL
LIN {X 0,Y 284.806,Z 521.627,A -85,B 0,C 180,E1 -17188.586,E2 -17188.586} C_VEL
LIN {X 0,Y 284.773,Z 521.852,A -85,B 0,C 180,E1 -17190,E2 -17190} C_VEL
LIN {X 0,Y 284.805,Z 521.665,A -85,B 0,C 180,E1 -17191.414,E2 -17191.414} C_VEL
LIN {X 0,Y 284.794,Z 521.111,A -85,B 0,C 180,E1 -17192.829,E2 -17192.829} C_VEL
LIN {X 0,Y 285.043,Z 520.159,A -85,B 0,C 180,E1 -17194.242,E2 -17194.242} C_VEL
LIN {X 0,Y 285.14,Z 518.86,A -85,B 0,C 180,E1 -17195.658,E2 -17195.658} C_VEL
LIN {X 0,Y 285.907,Z 516.031,A -85,B 0,C 180,E1 -17197.77,E2 -17197.77} C_VEL
LIN {X 0,Y 286.862,Z 512.201,A -85,B 0,C 180,E1 -17199.875,E2 -17199.875} C_VEL
LIN {X 0,Y 287.803,Z 507.118,A -85,B 0,C 180,E1 -17202.051,E2 -17202.051} C_VEL
LIN {X 0,Y 289.344,Z 499.875,A -85,B 0,C 180,E1 -17204.416,E2 -17204.416} C_VEL
LIN {X 0,Y 290.875,Z 491.844,A -85,B 0,C 180,E1 -17206.493,E2 -17206.493} C_VEL
LIN {X 0,Y 292.225,Z 483.618,A -85,B 0,C 180,E1 -17208.219,E2 -17208.219} C_VEL
LIN {X 0,Y 293.567,Z 474.583,A -85,B 0,C 180,E1 -17209.764,E2 -17209.764} C_VEL
LIN {X 0,Y 295.34,Z 463.032,A -85,B 0,C 180,E1 -17211.31,E2 -17211.31} C_VEL
LIN {X 0,Y 296.611,Z 451.099,A -85,B 0,C 180,E1 -17212.575,E2 -17212.575} C_VEL
LIN {X 0,Y 297.61,Z 438.504,A -85,B 0,C 180,E1 -17213.567,E2 -17213.567} C_VEL
LIN {X 0,Y 298.211,Z 425.9,A -85,B 0,C 180,E1 -17214.278,E2 -17214.278} C_VEL
LIN {X 0,Y 298.317,Z 416.029,A -85,B 0,C 180,E1 -17214.659,E2 -17214.659} C_VEL
LIN {X 0,Y 298.903,Z 379.079,A -85,B 0,C 180,E1 -17215.585,E2 -17215.585} C_VEL
LIN {X 0,Y 299.123,Z 367.516,A -85,B 0,C 180,E1 -17215.868,E2 -17215.868} C_VEL
LIN {X 0,Y 291.351,Z 350.436,A -85,B 0,C 180,E1 -17217.11,E2 -17217.11} C_VEL
LIN {X 0,Y 284.566,Z 337.171,A -85,B 0,C 180,E1 -17218.239,E2 -17218.239} C_VEL
LIN {X 0,Y 284.309,Z 336.178,A -85,B 0,C 180,E1 -17218.515,E2 -17218.515} C_VEL
LIN {X 0,Y 284.304,Z 336.056,A -85,B 0,C 180,E1 -17222.945,E2 -17222.945} C_VEL
LIN {X 0,Y 284.317,Z 336.052,A -85,B 0,C 180,E1 -17226.387,E2 -17226.387} C_VEL
LIN {X 0,Y 284.253,Z 336.078,A -85,B 0,C 180,E1 -17230.003,E2 -17230.003} C_VEL
LIN {X 0,Y 284.23,Z 336.054,A -85,B 0,C 180,E1 -17234.187,E2 -17234.187} C_VEL
LIN {X 0,Y 284.236,Z 336.071,A -85,B 0,C 180,E1 -17238.118,E2 -17238.118} C_VEL
LIN {X 0,Y 284.292,Z 336.035,A -85,B 0,C 180,E1 -17241.828,E2 -17241.828} C_VEL
LIN {X 0,Y 284.304,Z 336.07,A -85,B 0,C 180,E1 -17245.35,E2 -17245.35} C_VEL
LIN {X 0,Y 284.274,Z 336.033,A -85,B 0,C 180,E1 -17248.723,E2 -17248.723} C_VEL
LIN {X 0,Y 284.255,Z 336.031,A -85,B 0,C 180,E1 -17251.981,E2 -17251.981} C_VEL
LIN {X 0,Y 284.278,Z 336.073,A -85,B 0,C 180,E1 -17255.148,E2 -17255.148} C_VEL
LIN {X 0,Y 284.294,Z 336.059,A -85,B 0,C 180,E1 -17258.234,E2 -17258.234} C_VEL
LIN {X 0,Y 284.326,Z 336.066,A -85,B 0,C 180,E1 -17261.256,E2 -17261.256} C_VEL
LIN {X 0,Y 284.344,Z 336.063,A -85,B 0,C 180,E1 -17262.501,E2 -17262.501} C_VEL
LIN {X 0,Y 283.747,Z 336.142,A -85,B 0,C 180,E1 -17263.684,E2 -17263.684} C_VEL
LIN {X 0,Y 280.945,Z 336.494,A -85,B 0,C 180,E1 -17265.611,E2 -17265.611} C_VEL
LIN {X 0,Y 278.531,Z 336.792,A -85,B 0,C 180,E1 -17267.177,E2 -17267.177} C_VEL
LIN {X 0,Y 277.495,Z 336.919,A -85,B 0,C 180,E1 -17268.39,E2 -17268.39} C_VEL
LIN {X 0,Y 277.413,Z 336.926,A -85,B 0,C 180,E1 -17268.801,E2 -17268.801} C_VEL
LIN {X 0,Y 277.566,Z 336.895,A -85,B 0,C 180,E1 -17271.262,E2 -17271.262} C_VEL
LIN {X 0,Y 277.532,Z 336.908,A -85,B 0,C 180,E1 -17274.186,E2 -17274.186} C_VEL
LIN {X 0,Y 277.799,Z 336.861,A -85,B 0,C 180,E1 -17278.55,E2 -17278.55} C_VEL
LIN {X 0,Y 277.805,Z 336.875,A -85,B 0,C 180,E1 -17281.45,E2 -17281.45} C_VEL
LIN {X 0,Y 277.599,Z 336.893,A -85,B 0,C 180,E1 -17287.272,E2 -17287.272} C_VEL
LIN {X 0,Y 277.452,Z 336.923,A -85,B 0,C 180,E1 -17290.213,E2 -17290.213} C_VEL
LIN {X 0,Y 277.405,Z 336.924,A -85,B 0,C 180,E1 -17294.676,E2 -17294.676} C_VEL
LIN {X 0,Y 277.32,Z 336.914,A -85,B 0,C 180,E1 -17299.236,E2 -17299.236} C_VEL
LIN {X 0,Y 277.268,Z 336.944,A -85,B 0,C 180,E1 -17303.926,E2 -17303.926} C_VEL
LIN {X 0,Y 277.263,Z 336.926,A -85,B 0,C 180,E1 -17307.482,E2 -17307.482} C_VEL
LIN {X 0,Y 277.244,Z 336.943,A -85,B 0,C 180,E1 -17310.473,E2 -17310.473} C_VEL
LIN {X 0,Y 277.242,Z 336.934,A -85,B 0,C 180,E1 -17313.897,E2 -17313.897} C_VEL
LIN {X 0,Y 277.248,Z 336.951,A -85,B 0,C 180,E1 -17317.473,E2 -17317.473} C_VEL
LIN {X 0,Y 277.181,Z 336.959,A -85,B 0,C 180,E1 -17321.242,E2 -17321.242} C_VEL
LIN {X 0,Y 277.17,Z 336.917,A -85,B 0,C 180,E1 -17325.233,E2 -17325.233} C_VEL
LIN {X 0,Y 277.258,Z 337.176,A -85,B 0,C 180,E1 -17328.407,E2 -17328.407} C_VEL
LIN {X 0,Y 280.063,Z 347.514,A -85,B 0,C 180,E1 -17331.647,E2 -17331.647} C_VEL
LIN {X 0,Y 282.893,Z 359.287,A -85,B 0,C 180,E1 -17335.068,E2 -17335.068} C_VEL
LIN {X 0,Y 285.032,Z 369.977,A -85,B 0,C 180,E1 -17337.987,E2 -17337.987} C_VEL
LIN {X 0,Y 283.75,Z 378.198,A -85,B 0,C 180,E1 -17339.939,E2 -17339.939} C_VEL
LIN {X 0,Y 283.055,Z 382.732,A -85,B 0,C 180,E1 -17340.956,E2 -17340.956} C_VEL
LIN {X 0,Y 286.26,Z 406.706,A -85,B 0,C 180,E1 -17341.997,E2 -17341.997} C_VEL
LIN {X 0,Y 289.792,Z 440.125,A -85,B 0,C 180,E1 -17343.257,E2 -17343.257} C_VEL
LIN {X 0,Y 290.629,Z 453.31,A -85,B 0,C 180,E1 -17343.691,E2 -17343.691} C_VEL
LIN {X 0,Y 289.424,Z 494.53,A -85,B 0,C 180,E1 -17344.73,E2 -17344.73} C_VEL
LIN {X 0,Y 288.431,Z 508.234,A -85,B 0,C 180,E1 -17345.352,E2 -17345.352} C_VEL
LIN {X 0,Y 287.035,Z 520.532,A -85,B 0,C 180,E1 -17346.172,E2 -17346.172} C_VEL
LIN {X 0,Y 285.415,Z 531.713,A -85,B 0,C 180,E1 -17347.181,E2 -17347.181} C_VEL
LIN {X 0,Y 283.423,Z 543.377,A -85,B 0,C 180,E1 -17348.546,E2 -17348.546} C_VEL
LIN {X 0,Y 281.462,Z 553.911,A -85,B 0,C 180,E1 -17350.111,E2 -17350.111} C_VEL
LIN {X 0,Y 279.844,Z 562.564,A -85,B 0,C 180,E1 -17351.704,E2 -17351.704} C_VEL
LIN {X 0,Y 278.227,Z 571.431,A -85,B 0,C 180,E1 -17353.715,E2 -17353.715} C_VEL
LIN {X 0,Y 277.197,Z 578.482,A -85,B 0,C 180,E1 -17355.688,E2 -17355.688} C_VEL
LIN {X 0,Y 276.317,Z 585.813,A -85,B 0,C 180,E1 -17358.26,E2 -17358.26} C_VEL
LIN {X 0,Y 276.021,Z 590.741,A -85,B 0,C 180,E1 -17360.474,E2 -17360.474} C_VEL
LIN {X 0,Y 276.137,Z 595.062,A -85,B 0,C 180,E1 -17363.024,E2 -17363.024} C_VEL
LIN {X 0,Y 276.543,Z 598.049,A -85,B 0,C 180,E1 -17365.628,E2 -17365.628} C_VEL
LIN {X 0,Y 277.049,Z 599.809,A -85,B 0,C 180,E1 -17368.546,E2 -17368.546} C_VEL
LIN {X 0,Y 277.39,Z 600.08,A -85,B 0,C 180,E1 -17370,E2 -17370} C_VEL
LIN {X 0,Y 277.052,Z 599.801,A -85,B 0,C 180,E1 -17371.454,E2 -17371.454} C_VEL
LIN {X 0,Y 276.564,Z 598.036,A -85,B 0,C 180,E1 -17374.372,E2 -17374.372} C_VEL
LIN {X 0,Y 276.173,Z 594.946,A -85,B 0,C 180,E1 -17377.037,E2 -17377.037} C_VEL
LIN {X 0,Y 276.029,Z 590.69,A -85,B 0,C 180,E1 -17379.526,E2 -17379.526} C_VEL
LIN {X 0,Y 276.317,Z 585.746,A -85,B 0,C 180,E1 -17381.74,E2 -17381.74} C_VEL
LIN {X 0,Y 277.183,Z 578.398,A -85,B 0,C 180,E1 -17384.312,E2 -17384.312} C_VEL
LIN {X 0,Y 278.316,Z 571.084,A -85,B 0,C 180,E1 -17386.347,E2 -17386.347} C_VEL
LIN {X 0,Y 279.82,Z 562.426,A -85,B 0,C 180,E1 -17388.297,E2 -17388.297} C_VEL
LIN {X 0,Y 281.67,Z 552.664,A -85,B 0,C 180,E1 -17390.064,E2 -17390.064} C_VEL
LIN {X 0,Y 283.663,Z 541.875,A -85,B 0,C 180,E1 -17391.625,E2 -17391.625} C_VEL
LIN {X 0,Y 285.411,Z 531.467,A -85,B 0,C 180,E1 -17392.819,E2 -17392.819} C_VEL
LIN {X 0,Y 287.233,Z 519.054,A -85,B 0,C 180,E1 -17393.906,E2 -17393.906} C_VEL
LIN {X 0,Y 288.617,Z 505.705,A -85,B 0,C 180,E1 -17394.759,E2 -17394.759} C_VEL
LIN {X 0,Y 289.477,Z 493.134,A -85,B 0,C 180,E1 -17395.291,E2 -17395.291} C_VEL
LIN {X 0,Y 290.58,Z 450.682,A -85,B 0,C 180,E1 -17396.353,E2 -17396.353} C_VEL
LIN {X 0,Y 287.685,Z 419.665,A -85,B 0,C 180,E1 -17397.471,E2 -17397.471} C_VEL
LIN {X 0,Y 284.088,Z 390.398,A -85,B 0,C 180,E1 -17398.648,E2 -17398.648} C_VEL
LIN {X 0,Y 283.073,Z 382.649,A -85,B 0,C 180,E1 -17399.018,E2 -17399.018} C_VEL
LIN {X 0,Y 284.885,Z 371.475,A -85,B 0,C 180,E1 -17401.616,E2 -17401.616} C_VEL
LIN {X 0,Y 284.885,Z 368.781,A -85,B 0,C 180,E1 -17402.291,E2 -17402.291} C_VEL
LIN {X 0,Y 282.298,Z 356.584,A -85,B 0,C 180,E1 -17405.649,E2 -17405.649} C_VEL
LIN {X 0,Y 279.217,Z 344.169,A -85,B 0,C 180,E1 -17409.328,E2 -17409.328} C_VEL
LIN {X 0,Y 277.216,Z 337.024,A -85,B 0,C 180,E1 -17411.657,E2 -17411.657} C_VEL
LIN {X 0,Y 277.17,Z 336.918,A -85,B 0,C 180,E1 -17415.232,E2 -17415.232} C_VEL
LIN {X 0,Y 277.181,Z 336.96,A -85,B 0,C 180,E1 -17418.758,E2 -17418.758} C_VEL
LIN {X 0,Y 277.244,Z 336.879,A -85,B 0,C 180,E1 -17422.527,E2 -17422.527} C_VEL
LIN {X 0,Y 277.242,Z 336.929,A -85,B 0,C 180,E1 -17426.103,E2 -17426.103} C_VEL
LIN {X 0,Y 277.258,Z 336.94,A -85,B 0,C 180,E1 -17429.538,E2 -17429.538} C_VEL
LIN {X 0,Y 277.285,Z 336.928,A -85,B 0,C 180,E1 -17432.856,E2 -17432.856} C_VEL
LIN {X 0,Y 277.268,Z 336.944,A -85,B 0,C 180,E1 -17436.074,E2 -17436.074} C_VEL
LIN {X 0,Y 277.338,Z 336.913,A -85,B 0,C 180,E1 -17440.766,E2 -17440.766} C_VEL
LIN {X 0,Y 277.423,Z 336.921,A -85,B 0,C 180,E1 -17445.325,E2 -17445.325} C_VEL
LIN {X 0,Y 277.452,Z 336.924,A -85,B 0,C 180,E1 -17449.787,E2 -17449.787} C_VEL
LIN {X 0,Y 277.606,Z 336.892,A -85,B 0,C 180,E1 -17452.728,E2 -17452.728} C_VEL
LIN {X 0,Y 277.805,Z 336.876,A -85,B 0,C 180,E1 -17458.55,E2 -17458.55} C_VEL
LIN {X 0,Y 277.8,Z 336.86,A -85,B 0,C 180,E1 -17461.45,E2 -17461.45} C_VEL
LIN {X 0,Y 277.594,Z 336.888,A -85,B 0,C 180,E1 -17467.273,E2 -17467.273} C_VEL
LIN {X 0,Y 277.452,Z 336.922,A -85,B 0,C 180,E1 -17470.213,E2 -17470.213} C_VEL
LIN {X 0,Y 277.404,Z 336.908,A -85,B 0,C 180,E1 -17474.676,E2 -17474.676} C_VEL
LIN {X 0,Y 277.319,Z 336.935,A -85,B 0,C 180,E1 -17479.236,E2 -17479.236} C_VEL
LIN {X 0,Y 277.251,Z 336.95,A -85,B 0,C 180,E1 -17483.928,E2 -17483.928} C_VEL
LIN {X 0,Y 277.23,Z 336.916,A -85,B 0,C 180,E1 -17487.469,E2 -17487.469} C_VEL
LIN {X 0,Y 277.224,Z 336.897,A -85,B 0,C 180,E1 -17490.466,E2 -17490.466} C_VEL
LIN {X 0,Y 277.242,Z 336.949,A -85,B 0,C 180,E1 -17493.897,E2 -17493.897} C_VEL
LIN {X 0,Y 277.247,Z 336.922,A -85,B 0,C 180,E1 -17497.473,E2 -17497.473} C_VEL
LIN {X 0,Y 277.181,Z 336.936,A -85,B 0,C 180,E1 -17501.242,E2 -17501.242} C_VEL
LIN {X 0,Y 277.171,Z 336.941,A -85,B 0,C 180,E1 -17505.233,E2 -17505.233} C_VEL
LIN {X 0,Y 277.181,Z 336.946,A -85,B 0,C 180,E1 -17508.759,E2 -17508.759} C_VEL
LIN {X 0,Y 277.252,Z 336.926,A -85,B 0,C 180,E1 -17512.529,E2 -17512.529} C_VEL
LIN {X 0,Y 277.245,Z 336.943,A -85,B 0,C 180,E1 -17516.105,E2 -17516.105} C_VEL
LIN {X 0,Y 277.276,Z 336.988,A -85,B 0,C 180,E1 -17520.693,E2 -17520.693} C_VEL
LIN {X 0,Y 277.371,Z 337.59,A -85,B 0,C 180,E1 -17521.015,E2 -17521.015} C_VEL
LIN {X 0,Y 278.536,Z 340.209,A -85,B 0,C 180,E1 -17521.307,E2 -17521.307} C_VEL
LIN {X 0,Y 287.353,Z 357.335,A -85,B 0,C 180,E1 -17522.782,E2 -17522.782} C_VEL
LIN {X 0,Y 292.717,Z 369.285,A -85,B 0,C 180,E1 -17523.667,E2 -17523.667} C_VEL
LIN {X 0,Y 291.835,Z 416.811,A -85,B 0,C 180,E1 -17524.872,E2 -17524.872} C_VEL
LIN {X 0,Y 291.519,Z 430.019,A -85,B 0,C 180,E1 -17525.414,E2 -17525.414} C_VEL
LIN {X 0,Y 290.905,Z 441.54,A -85,B 0,C 180,E1 -17526.131,E2 -17526.131} C_VEL
LIN {X 0,Y 289.854,Z 453.786,A -85,B 0,C 180,E1 -17527.174,E2 -17527.174} C_VEL
LIN {X 0,Y 288.652,Z 464.052,A -85,B 0,C 180,E1 -17528.297,E2 -17528.297} C_VEL
LIN {X 0,Y 287.04,Z 474.801,A -85,B 0,C 180,E1 -17529.767,E2 -17529.767} C_VEL
LIN {X 0,Y 285.553,Z 483.995,A -85,B 0,C 180,E1 -17531.34,E2 -17531.34} C_VEL
LIN {X 0,Y 284.155,Z 492.346,A -85,B 0,C 180,E1 -17533.106,E2 -17533.106} C_VEL
LIN {X 0,Y 282.531,Z 500.463,A -85,B 0,C 180,E1 -17535.228,E2 -17535.228} C_VEL
LIN {X 0,Y 281.013,Z 507.571,A -85,B 0,C 180,E1 -17537.576,E2 -17537.576} C_VEL
LIN {X 0,Y 279.966,Z 512.944,A -85,B 0,C 180,E1 -17539.88,E2 -17539.88} C_VEL
LIN {X 0,Y 278.951,Z 516.835,A -85,B 0,C 180,E1 -17542.035,E2 -17542.035} C_VEL
LIN {X 0,Y 278.156,Z 519.711,A -85,B 0,C 180,E1 -17544.2,E2 -17544.2} C_VEL
LIN {X 0,Y 278.039,Z 521.05,A -85,B 0,C 180,E1 -17545.651,E2 -17545.651} C_VEL
LIN {X 0,Y 277.776,Z 522.027,A -85,B 0,C 180,E1 -17547.1,E2 -17547.1} C_VEL
LIN {X 0,Y 277.78,Z 522.605,A -85,B 0,C 180,E1 -17548.55,E2 -17548.55} C_VEL
LIN {X 0,Y 277.746,Z 522.83,A -85,B 0,C 180,E1 -17550,E2 -17550} C_VEL
LIN {X 0,Y 277.78,Z 522.643,A -85,B 0,C 180,E1 -17551.45,E2 -17551.45} C_VEL
LIN {X 0,Y 277.775,Z 522.089,A -85,B 0,C 180,E1 -17552.9,E2 -17552.9} C_VEL
LIN {X 0,Y 278.033,Z 521.137,A -85,B 0,C 180,E1 -17554.349,E2 -17554.349} C_VEL
LIN {X 0,Y 278.143,Z 519.838,A -85,B 0,C 180,E1 -17555.801,E2 -17555.801} C_VEL
LIN {X 0,Y 278.945,Z 517.008,A -85,B 0,C 180,E1 -17557.965,E2 -17557.965} C_VEL
LIN {X 0,Y 279.941,Z 513.178,A -85,B 0,C 180,E1 -17560.121,E2 -17560.121} C_VEL
LIN {X 0,Y 280.933,Z 508.095,A -85,B 0,C 180,E1 -17562.35,E2 -17562.35} C_VEL
LIN {X 0,Y 282.542,Z 500.851,A -85,B 0,C 180,E1 -17564.771,E2 -17564.771} C_VEL
LIN {X 0,Y 284.143,Z 492.82,A -85,B 0,C 180,E1 -17566.895,E2 -17566.895} C_VEL
LIN {X 0,Y 285.556,Z 484.594,A -85,B 0,C 180,E1 -17568.66,E2 -17568.66} C_VEL
LIN {X 0,Y 286.976,Z 475.555,A -85,B 0,C 180,E1 -17570.238,E2 -17570.238} C_VEL
LIN {X 0,Y 288.805,Z 464.005,A -85,B 0,C 180,E1 -17571.817,E2 -17571.817} C_VEL
LIN {X 0,Y 290.101,Z 452.387,A -85,B 0,C 180,E1 -17573.079,E2 -17573.079} C_VEL
LIN {X 0,Y 291.157,Z 440.625,A -85,B 0,C 180,E1 -17574.037,E2 -17574.037} C_VEL
LIN {X 0,Y 291.758,Z 427.89,A -85,B 0,C 180,E1 -17574.798,E2 -17574.798} C_VEL
LIN {X 0,Y 291.91,Z 417.392,A -85,B 0,C 180,E1 -17575.225,E2 -17575.225} C_VEL
LIN {X 0,Y 292.57,Z 379.136,A -85,B 0,C 180,E1 -17576.204,E2 -17576.204} C_VEL
LIN {X 0,Y 292.766,Z 369.362,A -85,B 0,C 180,E1 -17576.449,E2 -17576.449} C_VEL
LIN {X 0,Y 284.799,Z 352.035,A -85,B 0,C 180,E1 -17577.77,E2 -17577.77} C_VEL
LIN {X 0,Y 277.493,Z 338.106,A -85,B 0,C 180,E1 -17579.028,E2 -17579.028} C_VEL
LIN {X 0,Y 277.261,Z 337.055,A -85,B 0,C 180,E1 -17579.31,E2 -17579.31} C_VEL
LIN {X 0,Y 277.245,Z 336.942,A -85,B 0,C 180,E1 -17583.895,E2 -17583.895} C_VEL
LIN {X 0,Y 277.231,Z 336.929,A -85,B 0,C 180,E1 -17587.474,E2 -17587.474} C_VEL
LIN {X 0,Y 277.174,Z 336.949,A -85,B 0,C 180,E1 -17591.242,E2 -17591.242} C_VEL
LIN {X 0,Y 277.171,Z 336.947,A -85,B 0,C 180,E1 -17595.232,E2 -17595.232} C_VEL
LIN {X 0,Y 277.181,Z 336.939,A -85,B 0,C 180,E1 -17598.758,E2 -17598.758} C_VEL
LIN {X 0,Y 277.248,Z 336.921,A -85,B 0,C 180,E1 -17602.527,E2 -17602.527} C_VEL
LIN {X 0,Y 277.242,Z 336.949,A -85,B 0,C 180,E1 -17606.103,E2 -17606.103} C_VEL
LIN {X 0,Y 277.224,Z 336.898,A -85,B 0,C 180,E1 -17609.534,E2 -17609.534} C_VEL
LIN {X 0,Y 277.246,Z 336.918,A -85,B 0,C 180,E1 -17612.852,E2 -17612.852} C_VEL
LIN {X 0,Y 277.251,Z 336.95,A -85,B 0,C 180,E1 -17616.072,E2 -17616.072} C_VEL
LIN {X 0,Y 277.279,Z 336.94,A -85,B 0,C 180,E1 -17620.761,E2 -17620.761} C_VEL
LIN {X 0,Y 277.404,Z 336.909,A -85,B 0,C 180,E1 -17625.324,E2 -17625.324} C_VEL
LIN {X 0,Y 277.413,Z 336.926,A -85,B 0,C 180,E1 -17628.801,E2 -17628.801} C_VEL
LIN {X 0,Y 276.761,Z 337.006,A -85,B 0,C 180,E1 -17630.014,E2 -17630.014} C_VEL
LIN {X 0,Y 273.946,Z 337.348,A -85,B 0,C 180,E1 -17631.992,E2 -17631.992} C_VEL
LIN {X 0,Y 271.539,Z 337.651,A -85,B 0,C 180,E1 -17633.599,E2 -17633.599} C_VEL
LIN {X 0,Y 270.487,Z 337.792,A -85,B 0,C 180,E1 -17634.843,E2 -17634.843} C_VEL
LIN {X 0,Y 270.39,Z 337.8,A -85,B 0,C 180,E1 -17635.265,E2 -17635.265} C_VEL
LIN {X 0,Y 270.765,Z 337.737,A -85,B 0,C 180,E1 -17638.513,E2 -17638.513} C_VEL
LIN {X 0,Y 270.769,Z 337.752,A -85,B 0,C 180,E1 -17641.487,E2 -17641.487} C_VEL
LIN {X 0,Y 270.56,Z 337.771,A -85,B 0,C 180,E1 -17647.463,E2 -17647.463} C_VEL
LIN {X 0,Y 270.404,Z 337.798,A -85,B 0,C 180,E1 -17650.482,E2 -17650.482} C_VEL
LIN {X 0,Y 270.373,Z 337.804,A -85,B 0,C 180,E1 -17655.066,E2 -17655.066} C_VEL
LIN {X 0,Y 270.256,Z 337.787,A -85,B 0,C 180,E1 -17659.759,E2 -17659.759} C_VEL
LIN {X 0,Y 270.194,Z 337.829,A -85,B 0,C 180,E1 -17664.593,E2 -17664.593} C_VEL
LIN {X 0,Y 270.192,Z 337.803,A -85,B 0,C 180,E1 -17667.918,E2 -17667.918} C_VEL
LIN {X 0,Y 270.17,Z 337.831,A -85,B 0,C 180,E1 -17671.35,E2 -17671.35} C_VEL
LIN {X 0,Y 270.194,Z 337.81,A -85,B 0,C 180,E1 -17674.907,E2 -17674.907} C_VEL
LIN {X 0,Y 270.195,Z 337.816,A -85,B 0,C 180,E1 -17678.711,E2 -17678.711} C_VEL
LIN {X 0,Y 270.144,Z 337.806,A -85,B 0,C 180,E1 -17683.245,E2 -17683.245} C_VEL
LIN {X 0,Y 270.19,Z 337.986,A -85,B 0,C 180,E1 -17687.62,E2 -17687.62} C_VEL
LIN {X 0,Y 273.099,Z 348.686,A -85,B 0,C 180,E1 -17691.119,E2 -17691.119} C_VEL
LIN {X 0,Y 275.938,Z 360.213,A -85,B 0,C 180,E1 -17694.59,E2 -17694.59} C_VEL
LIN {X 0,Y 278.124,Z 370.858,A -85,B 0,C 180,E1 -17697.602,E2 -17697.602} C_VEL
LIN {X 0,Y 277.629,Z 375.434,A -85,B 0,C 180,E1 -17698.739,E2 -17698.739} C_VEL
LIN {X 0,Y 276.479,Z 381.596,A -85,B 0,C 180,E1 -17700.183,E2 -17700.183} C_VEL
LIN {X 0,Y 279.319,Z 402.557,A -85,B 0,C 180,E1 -17701.15,E2 -17701.15} C_VEL
LIN {X 0,Y 282.961,Z 435.956,A -85,B 0,C 180,E1 -17702.472,E2 -17702.472} C_VEL
LIN {X 0,Y 284.238,Z 453.096,A -85,B 0,C 180,E1 -17703.073,E2 -17703.073} C_VEL
LIN {X 0,Y 283.018,Z 493.26,A -85,B 0,C 180,E1 -17704.104,E2 -17704.104} C_VEL
LIN {X 0,Y 282.066,Z 506.67,A -85,B 0,C 180,E1 -17704.719,E2 -17704.719} C_VEL
LIN {X 0,Y 280.522,Z 519.545,A -85,B 0,C 180,E1 -17705.583,E2 -17705.583} C_VEL
LIN {X 0,Y 278.878,Z 530.729,A -85,B 0,C 180,E1 -17706.615,E2 -17706.615} C_VEL
LIN {X 0,Y 276.817,Z 542.391,A -85,B 0,C 180,E1 -17708.008,E2 -17708.008} C_VEL
LIN {X 0,Y 274.785,Z 552.925,A -85,B 0,C 180,E1 -17709.606,E2 -17709.606} C_VEL
LIN {X 0,Y 273.056,Z 561.57,A -85,B 0,C 180,E1 -17711.233,E2 -17711.233} C_VEL
LIN {X 0,Y 271.606,Z 569.602,A -85,B 0,C 180,E1 -17713.076,E2 -17713.076} C_VEL
LIN {X 0,Y 270.676,Z 574.539,A -85,B 0,C 180,E1 -17714.421,E2 -17714.421} C_VEL
LIN {X 0,Y 269.658,Z 581.898,A -85,B 0,C 180,E1 -17716.818,E2 -17716.818} C_VEL
LIN {X 0,Y 269.035,Z 588.245,A -85,B 0,C 180,E1 -17719.464,E2 -17719.464} C_VEL
LIN {X 0,Y 268.942,Z 592.419,A -85,B 0,C 180,E1 -17721.737,E2 -17721.737} C_VEL
LIN {X 0,Y 269.173,Z 595.547,A -85,B 0,C 180,E1 -17724.005,E2 -17724.005} C_VEL
LIN {X 0,Y 269.463,Z 597.061,A -85,B 0,C 180,E1 -17725.512,E2 -17725.512} C_VEL
LIN {X 0,Y 269.678,Z 598.143,A -85,B 0,C 180,E1 -17727.012,E2 -17727.012} C_VEL
LIN {X 0,Y 269.989,Z 598.826,A -85,B 0,C 180,E1 -17728.508,E2 -17728.508} C_VEL
LIN {X 0,Y 270.353,Z 599.101,A -85,B 0,C 180,E1 -17730,E2 -17730} C_VEL
LIN {X 0,Y 269.993,Z 598.818,A -85,B 0,C 180,E1 -17731.492,E2 -17731.492} C_VEL
LIN {X 0,Y 269.689,Z 598.131,A -85,B 0,C 180,E1 -17732.987,E2 -17732.987} C_VEL
LIN {X 0,Y 269.483,Z 597.047,A -85,B 0,C 180,E1 -17734.487,E2 -17734.487} C_VEL
LIN {X 0,Y 269.11,Z 594.165,A -85,B 0,C 180,E1 -17737.069,E2 -17737.069} C_VEL
LIN {X 0,Y 268.964,Z 589.692,A -85,B 0,C 180,E1 -17739.779,E2 -17739.779} C_VEL
LIN {X 0,Y 269.3,Z 584.746,A -85,B 0,C 180,E1 -17742.051,E2 -17742.051} C_VEL
LIN {X 0,Y 270.271,Z 577.403,A -85,B 0,C 180,E1 -17744.686,E2 -17744.686} C_VEL
LIN {X 0,Y 271.33,Z 570.774,A -85,B 0,C 180,E1 -17746.589,E2 -17746.589} C_VEL
LIN {X 0,Y 273.035,Z 561.427,A -85,B 0,C 180,E1 -17748.769,E2 -17748.769} C_VEL
LIN {X 0,Y 275.019,Z 551.673,A -85,B 0,C 180,E1 -17750.571,E2 -17750.571} C_VEL
LIN {X 0,Y 277.036,Z 540.877,A -85,B 0,C 180,E1 -17752.17,E2 -17752.17} C_VEL
LIN {X 0,Y 278.875,Z 530.474,A -85,B 0,C 180,E1 -17753.385,E2 -17753.385} C_VEL
LIN {X 0,Y 280.753,Z 518.059,A -85,B 0,C 180,E1 -17754.494,E2 -17754.494} C_VEL
LIN {X 0,Y 282.119,Z 504.87,A -85,B 0,C 180,E1 -17755.358,E2 -17755.358} C_VEL
LIN {X 0,Y 283.072,Z 491.836,A -85,B 0,C 180,E1 -17755.916,E2 -17755.916} C_VEL
LIN {X 0,Y 284.133,Z 451.058,A -85,B 0,C 180,E1 -17756.96,E2 -17756.96} C_VEL
LIN {X 0,Y 281.393,Z 420.956,A -85,B 0,C 180,E1 -17758.074,E2 -17758.074} C_VEL
LIN {X 0,Y 277.973,Z 392.597,A -85,B 0,C 180,E1 -17759.247,E2 -17759.247} C_VEL
LIN {X 0,Y 276.512,Z 381.713,A -85,B 0,C 180,E1 -17759.762,E2 -17759.762} C_VEL
LIN {X 0,Y 278.102,Z 372.074,A -85,B 0,C 180,E1 -17762.052,E2 -17762.052} C_VEL
LIN {X 0,Y 277.362,Z 366.901,A -85,B 0,C 180,E1 -17763.46,E2 -17763.46} C_VEL
LIN {X 0,Y 274.566,Z 354.534,A -85,B 0,C 180,E1 -17767.04,E2 -17767.04} C_VEL
LIN {X 0,Y 271.559,Z 342.94,A -85,B 0,C 180,E1 -17770.665,E2 -17770.665} C_VEL
LIN {X 0,Y 270.162,Z 337.913,A -85,B 0,C 180,E1 -17772.405,E2 -17772.405} C_VEL
LIN {X 0,Y 270.144,Z 337.808,A -85,B 0,C 180,E1 -17776.755,E2 -17776.755} C_VEL
LIN {X 0,Y 270.195,Z 337.769,A -85,B 0,C 180,E1 -17781.289,E2 -17781.289} C_VEL
LIN {X 0,Y 270.193,Z 337.778,A -85,B 0,C 180,E1 -17785.093,E2 -17785.093} C_VEL
LIN {X 0,Y 270.18,Z 337.827,A -85,B 0,C 180,E1 -17789.136,E2 -17789.136} C_VEL
LIN {X 0,Y 270.195,Z 337.804,A -85,B 0,C 180,E1 -17792.172,E2 -17792.172} C_VEL
LIN {X 0,Y 270.213,Z 337.828,A -85,B 0,C 180,E1 -17795.547,E2 -17795.547} C_VEL
LIN {X 0,Y 270.284,Z 337.784,A -85,B 0,C 180,E1 -17800.243,E2 -17800.243} C_VEL
LIN {X 0,Y 270.392,Z 337.801,A -85,B 0,C 180,E1 -17804.935,E2 -17804.935} C_VEL
LIN {X 0,Y 270.405,Z 337.799,A -85,B 0,C 180,E1 -17809.518,E2 -17809.518} C_VEL
LIN {X 0,Y 270.566,Z 337.771,A -85,B 0,C 180,E1 -17812.538,E2 -17812.538} C_VEL
LIN {X 0,Y 270.769,Z 337.752,A -85,B 0,C 180,E1 -17818.513,E2 -17818.513} C_VEL
LIN {X 0,Y 270.765,Z 337.736,A -85,B 0,C 180,E1 -17821.487,E2 -17821.487} C_VEL
LIN {X 0,Y 270.556,Z 337.763,A -85,B 0,C 180,E1 -17827.463,E2 -17827.463} C_VEL
LIN {X 0,Y 270.405,Z 337.799,A -85,B 0,C 180,E1 -17830.483,E2 -17830.483} C_VEL
LIN {X 0,Y 270.372,Z 337.785,A -85,B 0,C 180,E1 -17835.067,E2 -17835.067} C_VEL
LIN {X 0,Y 270.256,Z 337.808,A -85,B 0,C 180,E1 -17839.759,E2 -17839.759} C_VEL
LIN {X 0,Y 270.173,Z 337.83,A -85,B 0,C 180,E1 -17844.596,E2 -17844.596} C_VEL
LIN {X 0,Y 270.18,Z 337.783,A -85,B 0,C 180,E1 -17847.919,E2 -17847.919} C_VEL
LIN {X 0,Y 270.165,Z 337.787,A -85,B 0,C 180,E1 -17851.351,E2 -17851.351} C_VEL
LIN {X 0,Y 270.194,Z 337.829,A -85,B 0,C 180,E1 -17854.907,E2 -17854.907} C_VEL
LIN {X 0,Y 270.195,Z 337.785,A -85,B 0,C 180,E1 -17858.711,E2 -17858.711} C_VEL
LIN {X 0,Y 270.145,Z 337.836,A -85,B 0,C 180,E1 -17863.246,E2 -17863.246} C_VEL
LIN {X 0,Y 270.148,Z 337.804,A -85,B 0,C 180,E1 -17867.438,E2 -17867.438} C_VEL
LIN {X 0,Y 270.206,Z 337.813,A -85,B 0,C 180,E1 -17871.375,E2 -17871.375} C_VEL
LIN {X 0,Y 270.197,Z 337.829,A -85,B 0,C 180,E1 -17875.095,E2 -17875.095} C_VEL
LIN {X 0,Y 270.171,Z 337.83,A -85,B 0,C 180,E1 -17879.142,E2 -17879.142} C_VEL
LIN {X 0,Y 270.254,Z 338.104,A -85,B 0,C 180,E1 -17880.068,E2 -17880.068} C_VEL
LIN {X 0,Y 270.521,Z 339.17,A -85,B 0,C 180,E1 -17880.288,E2 -17880.288} C_VEL
LIN {X 0,Y 280.313,Z 357.795,A -85,B 0,C 180,E1 -17882.02,E2 -17882.02} C_VEL
LIN {X 0,Y 286.399,Z 371.27,A -85,B 0,C 180,E1 -17883.067,E2 -17883.067} C_VEL
LIN {X 0,Y 285.49,Z 417.464,A -85,B 0,C 180,E1 -17884.262,E2 -17884.262} C_VEL
LIN {X 0,Y 285.121,Z 431.197,A -85,B 0,C 180,E1 -17884.835,E2 -17884.835} C_VEL
LIN {X 0,Y 284.424,Z 443.672,A -85,B 0,C 180,E1 -17885.649,E2 -17885.649} C_VEL
LIN {X 0,Y 283.225,Z 456.498,A -85,B 0,C 180,E1 -17886.8,E2 -17886.8} C_VEL
LIN {X 0,Y 281.765,Z 467.16,A -85,B 0,C 180,E1 -17888.029,E2 -17888.029} C_VEL
LIN {X 0,Y 280.048,Z 477.995,A -85,B 0,C 180,E1 -17889.623,E2 -17889.623} C_VEL
LIN {X 0,Y 278.581,Z 486.76,A -85,B 0,C 180,E1 -17891.237,E2 -17891.237} C_VEL
LIN {X 0,Y 277.135,Z 494.782,A -85,B 0,C 180,E1 -17893.045,E2 -17893.045} C_VEL
LIN {X 0,Y 275.506,Z 502.642,A -85,B 0,C 180,E1 -17895.221,E2 -17895.221} C_VEL
LIN {X 0,Y 274.154,Z 508.551,A -85,B 0,C 180,E1 -17897.26,E2 -17897.26} C_VEL
LIN {X 0,Y 273.05,Z 513.923,A -85,B 0,C 180,E1 -17899.62,E2 -17899.62} C_VEL
LIN {X 0,Y 271.993,Z 517.814,A -85,B 0,C 180,E1 -17901.83,E2 -17901.83} C_VEL
LIN {X 0,Y 271.161,Z 520.69,A -85,B 0,C 180,E1 -17904.049,E2 -17904.049} C_VEL
LIN {X 0,Y 271.03,Z 522.029,A -85,B 0,C 180,E1 -17905.538,E2 -17905.538} C_VEL
LIN {X 0,Y 270.757,Z 523.005,A -85,B 0,C 180,E1 -17907.024,E2 -17907.024} C_VEL
LIN {X 0,Y 270.755,Z 523.583,A -85,B 0,C 180,E1 -17908.513,E2 -17908.513} C_VEL
LIN {X 0,Y 270.719,Z 523.808,A -85,B 0,C 180,E1 -17910,E2 -17910} C_VEL
LIN {X 0,Y 270.755,Z 523.621,A -85,B 0,C 180,E1 -17911.487,E2 -17911.487} C_VEL
LIN {X 0,Y 270.756,Z 523.066,A -85,B 0,C 180,E1 -17912.976,E2 -17912.976} C_VEL
LIN {X 0,Y 271.024,Z 522.115,A -85,B 0,C 180,E1 -17914.462,E2 -17914.462} C_VEL
LIN {X 0,Y 271.148,Z 520.815,A -85,B 0,C 180,E1 -17915.951,E2 -17915.951} C_VEL
LIN {X 0,Y 271.987,Z 517.985,A -85,B 0,C 180,E1 -17918.17,E2 -17918.17} C_VEL
LIN {X 0,Y 273.025,Z 514.154,A -85,B 0,C 180,E1 -17920.381,E2 -17920.381} C_VEL
LIN {X 0,Y 274.072,Z 509.071,A -85,B 0,C 180,E1 -17922.664,E2 -17922.664} C_VEL
LIN {X 0,Y 275.752,Z 501.827,A -85,B 0,C 180,E1 -17925.143,E2 -17925.143} C_VEL
LIN {X 0,Y 277.425,Z 493.795,A -85,B 0,C 180,E1 -17927.317,E2 -17927.317} C_VEL
LIN {X 0,Y 278.904,Z 485.569,A -85,B 0,C 180,E1 -17929.122,E2 -17929.122} C_VEL
LIN {X 0,Y 280.395,Z 476.529,A -85,B 0,C 180,E1 -17930.734,E2 -17930.734} C_VEL
LIN {X 0,Y 282.302,Z 464.976,A -85,B 0,C 180,E1 -17932.346,E2 -17932.346} C_VEL
LIN {X 0,Y 283.65,Z 453.358,A -85,B 0,C 180,E1 -17933.635,E2 -17933.635} C_VEL
LIN {X 0,Y 284.746,Z 441.595,A -85,B 0,C 180,E1 -17934.613,E2 -17934.613} C_VEL
LIN {X 0,Y 285.366,Z 429.859,A -85,B 0,C 180,E1 -17935.338,E2 -17935.338} C_VEL
LIN {X 0,Y 285.535,Z 418.237,A -85,B 0,C 180,E1 -17935.833,E2 -17935.833} C_VEL
LIN {X 0,Y 286.322,Z 377.99,A -85,B 0,C 180,E1 -17936.879,E2 -17936.879} C_VEL
LIN {X 0,Y 286.439,Z 371.248,A -85,B 0,C 180,E1 -17937.054,E2 -17937.054} C_VEL
LIN {X 0,Y 278.34,Z 353.795,A -85,B 0,C 180,E1 -17938.45,E2 -17938.45} C_VEL
LIN {X 0,Y 270.424,Z 338.862,A -85,B 0,C 180,E1 -17939.879,E2 -17939.879} C_VEL
LIN {X 0,Y 270.217,Z 337.872,A -85,B 0,C 180,E1 -17940.206,E2 -17940.206} C_VEL
LIN {X 0,Y 270.214,Z 337.814,A -85,B 0,C 180,E1 -17943.665,E2 -17943.665} C_VEL
LIN {X 0,Y 270.197,Z 337.807,A -85,B 0,C 180,E1 -17946.744,E2 -17946.744} C_VEL
LIN {X 0,Y 270.132,Z 337.83,A -85,B 0,C 180,E1 -17951.019,E2 -17951.019} C_VEL
LIN {X 0,Y 270.126,Z 337.815,A -85,B 0,C 180,E1 -17954.625,E2 -17954.625} C_VEL
LIN {X 0,Y 270.148,Z 337.834,A -85,B 0,C 180,E1 -17957.437,E2 -17957.437} C_VEL
LIN {X 0,Y 270.189,Z 337.786,A -85,B 0,C 180,E1 -17961.371,E2 -17961.371} C_VEL
LIN {X 0,Y 270.194,Z 337.829,A -85,B 0,C 180,E1 -17965.093,E2 -17965.093} C_VEL
LIN {X 0,Y 270.167,Z 337.78,A -85,B 0,C 180,E1 -17969.141,E2 -17969.141} C_VEL
LIN {X 0,Y 270.183,Z 337.784,A -85,B 0,C 180,E1 -17972.177,E2 -17972.177} C_VEL
LIN {X 0,Y 270.178,Z 337.829,A -85,B 0,C 180,E1 -17975.564,E2 -17975.564} C_VEL
LIN {X 0,Y 270.218,Z 337.813,A -85,B 0,C 180,E1 -17980.238,E2 -17980.238} C_VEL
LIN {X 0,Y 270.363,Z 337.787,A -85,B 0,C 180,E1 -17984.933,E2 -17984.933} C_VEL
LIN {X 0,Y 270.405,Z 337.8,A -85,B 0,C 180,E1 -17989.517,E2 -17989.517} C_VEL
LIN {X 0,Y 270.555,Z 337.764,A -85,B 0,C 180,E1 -17992.537,E2 -17992.537} C_VEL
LIN {X 0,Y 270.39,Z 337.8,A -85,B 0,C 180,E1 -17995.265,E2 -17995.265} C_VEL
LIN {X 0,Y 269.762,Z 337.887,A -85,B 0,C 180,E1 -17996.511,E2 -17996.511} C_VEL
LIN {X 0,Y 267.152,Z 338.214,A -85,B 0,C 180,E1 -17998.549,E2 -17998.549} C_VEL
LIN {X 0,Y 264.065,Z 338.588,A -85,B 0,C 180,E1 -18001.049,E2 -18001.049} C_VEL
LIN {X 0,Y 263.659,Z 338.636,A -85,B 0,C 180,E1 -18001.911,E2 -18001.911} C_VEL
LIN {X 0,Y 263.524,Z 338.649,A -85,B 0,C 180,E1 -18007.663,E2 -18007.663} C_VEL
LIN {X 0,Y 263.344,Z 338.675,A -85,B 0,C 180,E1 -18010.767,E2 -18010.767} C_VEL
LIN {X 0,Y 263.319,Z 338.683,A -85,B 0,C 180,E1 -18015.48,E2 -18015.48} C_VEL
LIN {X 0,Y 263.233,Z 338.657,A -85,B 0,C 180,E1 -18020.309,E2 -18020.309} C_VEL
LIN {X 0,Y 263.132,Z 338.708,A -85,B 0,C 180,E1 -18025.299,E2 -18025.299} C_VEL
LIN {X 0,Y 263.129,Z 338.682,A -85,B 0,C 180,E1 -18028.736,E2 -18028.736} C_VEL
LIN {X 0,Y 263.124,Z 338.708,A -85,B 0,C 180,E1 -18032.289,E2 -18032.289} C_VEL
LIN {X 0,Y 263.17,Z 338.704,A -85,B 0,C 180,E1 -18036.761,E2 -18036.761} C_VEL
LIN {X 0,Y 263.088,Z 338.7,A -85,B 0,C 180,E1 -18039.876,E2 -18039.876} C_VEL
LIN {X 0,Y 263.073,Z 338.676,A -85,B 0,C 180,E1 -18043.995,E2 -18043.995} C_VEL
LIN {X 0,Y 263.128,Z 338.877,A -85,B 0,C 180,E1 -18046.845,E2 -18046.845} C_VEL
LIN {X 0,Y 266.263,Z 350.24,A -85,B 0,C 180,E1 -18050.694,E2 -18050.694} C_VEL
LIN {X 0,Y 269.2,Z 362.358,A -85,B 0,C 180,E1 -18054.453,E2 -18054.453} C_VEL
LIN {X 0,Y 271.279,Z 372.79,A -85,B 0,C 180,E1 -18057.482,E2 -18057.482} C_VEL
LIN {X 0,Y 269.991,Z 380.375,A -85,B 0,C 180,E1 -18059.359,E2 -18059.359} C_VEL
LIN {X 0,Y 270.565,Z 385.398,A -85,B 0,C 180,E1 -18059.653,E2 -18059.653} C_VEL
LIN {X 0,Y 273.458,Z 406.878,A -85,B 0,C 180,E1 -18060.624,E2 -18060.624} C_VEL
LIN {X 0,Y 276.914,Z 440.048,A -85,B 0,C 180,E1 -18061.961,E2 -18061.961} C_VEL
LIN {X 0,Y 277.862,Z 453.829,A -85,B 0,C 180,E1 -18062.452,E2 -18062.452} C_VEL
LIN {X 0,Y 276.674,Z 492.082,A -85,B 0,C 180,E1 -18063.455,E2 -18063.455} C_VEL
LIN {X 0,Y 275.611,Z 505.809,A -85,B 0,C 180,E1 -18064.092,E2 -18064.092} C_VEL
LIN {X 0,Y 274.036,Z 518.558,A -85,B 0,C 180,E1 -18064.966,E2 -18064.966} C_VEL
LIN {X 0,Y 272.375,Z 529.745,A -85,B 0,C 180,E1 -18066.022,E2 -18066.022} C_VEL
LIN {X 0,Y 270.197,Z 541.399,A -85,B 0,C 180,E1 -18067.44,E2 -18067.44} C_VEL
LIN {X 0,Y 268.138,Z 551.94,A -85,B 0,C 180,E1 -18069.077,E2 -18069.077} C_VEL
LIN {X 0,Y 266.29,Z 560.577,A -85,B 0,C 180,E1 -18070.737,E2 -18070.737} C_VEL
LIN {X 0,Y 264.777,Z 568.61,A -85,B 0,C 180,E1 -18072.626,E2 -18072.626} C_VEL
LIN {X 0,Y 263.695,Z 573.893,A -85,B 0,C 180,E1 -18074.108,E2 -18074.108} C_VEL
LIN {X 0,Y 262.665,Z 580.899,A -85,B 0,C 180,E1 -18076.461,E2 -18076.461} C_VEL
LIN {X 0,Y 261.984,Z 587.248,A -85,B 0,C 180,E1 -18079.177,E2 -18079.177} C_VEL
LIN {X 0,Y 261.887,Z 591.428,A -85,B 0,C 180,E1 -18081.512,E2 -18081.512} C_VEL
LIN {X 0,Y 262.094,Z 594.557,A -85,B 0,C 180,E1 -18083.843,E2 -18083.843} C_VEL
LIN {X 0,Y 262.385,Z 596.074,A -85,B 0,C 180,E1 -18085.391,E2 -18085.391} C_VEL
LIN {X 0,Y 262.616,Z 597.159,A -85,B 0,C 180,E1 -18086.932,E2 -18086.932} C_VEL
LIN {X 0,Y 262.928,Z 597.843,A -85,B 0,C 180,E1 -18088.468,E2 -18088.468} C_VEL
LIN {X 0,Y 263.316,Z 598.122,A -85,B 0,C 180,E1 -18090,E2 -18090} C_VEL
LIN {X 0,Y 262.932,Z 597.835,A -85,B 0,C 180,E1 -18091.532,E2 -18091.532} C_VEL
LIN {X 0,Y 262.627,Z 597.147,A -85,B 0,C 180,E1 -18093.068,E2 -18093.068} C_VEL
LIN {X 0,Y 262.405,Z 596.058,A -85,B 0,C 180,E1 -18094.609,E2 -18094.609} C_VEL
LIN {X 0,Y 262.041,Z 593.382,A -85,B 0,C 180,E1 -18097.092,E2 -18097.092} C_VEL
LIN {X 0,Y 261.871,Z 590.084,A -85,B 0,C 180,E1 -18099.266,E2 -18099.266} C_VEL
LIN {X 0,Y 262.114,Z 585.521,A -85,B 0,C 180,E1 -18101.601,E2 -18101.601} C_VEL
LIN {X 0,Y 262.811,Z 579.774,A -85,B 0,C 180,E1 -18103.926,E2 -18103.926} C_VEL
LIN {X 0,Y 263.879,Z 572.358,A -85,B 0,C 180,E1 -18106.325,E2 -18106.325} C_VEL
LIN {X 0,Y 265.316,Z 565.443,A -85,B 0,C 180,E1 -18108.134,E2 -18108.134} C_VEL
LIN {X 0,Y 267.066,Z 556.789,A -85,B 0,C 180,E1 -18110.005,E2 -18110.005} C_VEL
LIN {X 0,Y 269.268,Z 546.161,A -85,B 0,C 180,E1 -18111.834,E2 -18111.834} C_VEL
LIN {X 0,Y 271.282,Z 535.676,A -85,B 0,C 180,E1 -18113.27,E2 -18113.27} C_VEL
LIN {X 0,Y 273.24,Z 524.201,A -85,B 0,C 180,E1 -18114.503,E2 -18114.503} C_VEL
LIN {X 0,Y 274.837,Z 512.394,A -85,B 0,C 180,E1 -18115.462,E2 -18115.462} C_VEL
LIN {X 0,Y 276.119,Z 498.964,A -85,B 0,C 180,E1 -18116.237,E2 -18116.237} C_VEL
LIN {X 0,Y 276.887,Z 485.551,A -85,B 0,C 180,E1 -18116.716,E2 -18116.716} C_VEL
LIN {X 0,Y 277.803,Z 452.171,A -85,B 0,C 180,E1 -18117.566,E2 -18117.566} C_VEL
LIN {X 0,Y 274.77,Z 418.415,A -85,B 0,C 180,E1 -18118.856,E2 -18118.856} C_VEL
LIN {X 0,Y 270.763,Z 386.546,A -85,B 0,C 180,E1 -18120.25,E2 -18120.25} C_VEL
LIN {X 0,Y 270.008,Z 380.51,A -85,B 0,C 180,E1 -18120.581,E2 -18120.581} C_VEL
LIN {X 0,Y 271.237,Z 372.646,A -85,B 0,C 180,E1 -18122.523,E2 -18122.523} C_VEL
LIN {X 0,Y 269.154,Z 362.233,A -85,B 0,C 180,E1 -18125.542,E2 -18125.542} C_VEL
LIN {X 0,Y 266.573,Z 351.62,A -85,B 0,C 180,E1 -18128.819,E2 -18128.819} C_VEL
LIN {X 0,Y 263.892,Z 341.683,A -85,B 0,C 180,E1 -18132.111,E2 -18132.111} C_VEL
LIN {X 0,Y 263.134,Z 338.79,A -85,B 0,C 180,E1 -18133.192,E2 -18133.192} C_VEL
LIN {X 0,Y 263.075,Z 338.679,A -85,B 0,C 180,E1 -18136.161,E2 -18136.161} C_VEL
LIN {X 0,Y 263.088,Z 338.679,A -85,B 0,C 180,E1 -18140.124,E2 -18140.124} C_VEL
LIN {X 0,Y 263.151,Z 338.636,A -85,B 0,C 180,E1 -18144.016,E2 -18144.016} C_VEL
LIN {X 0,Y 263.124,Z 338.708,A -85,B 0,C 180,E1 -18147.711,E2 -18147.711} C_VEL
LIN {X 0,Y 263.142,Z 338.68,A -85,B 0,C 180,E1 -18151.805,E2 -18151.805} C_VEL
LIN {X 0,Y 263.134,Z 338.702,A -85,B 0,C 180,E1 -18156.382,E2 -18156.382} C_VEL
LIN {X 0,Y 263.245,Z 338.656,A -85,B 0,C 180,E1 -18159.692,E2 -18159.692} C_VEL
LIN {X 0,Y 263.34,Z 338.68,A -85,B 0,C 180,E1 -18164.521,E2 -18164.521} C_VEL
LIN {X 0,Y 263.345,Z 338.677,A -85,B 0,C 180,E1 -18169.233,E2 -18169.233} C_VEL
LIN {X 0,Y 263.528,Z 338.648,A -85,B 0,C 180,E1 -18172.337,E2 -18172.337} C_VEL
LIN {X 0,Y 263.733,Z 338.629,A -85,B 0,C 180,E1 -18178.473,E2 -18178.473} C_VEL
LIN {X 0,Y 263.729,Z 338.613,A -85,B 0,C 180,E1 -18181.527,E2 -18181.527} C_VEL
LIN {X 0,Y 263.52,Z 338.638,A -85,B 0,C 180,E1 -18187.663,E2 -18187.663} C_VEL
LIN {X 0,Y 263.344,Z 338.679,A -85,B 0,C 180,E1 -18190.767,E2 -18190.767} C_VEL
LIN {X 0,Y 263.319,Z 338.666,A -85,B 0,C 180,E1 -18195.48,E2 -18195.48} C_VEL
LIN {X 0,Y 263.233,Z 338.679,A -85,B 0,C 180,E1 -18200.309,E2 -18200.309} C_VEL
LIN {X 0,Y 263.116,Z 338.704,A -85,B 0,C 180,E1 -18205.301,E2 -18205.301} C_VEL
LIN {X 0,Y 263.114,Z 338.652,A -85,B 0,C 180,E1 -18208.738,E2 -18208.738} C_VEL
LIN {X 0,Y 263.123,Z 338.681,A -85,B 0,C 180,E1 -18212.29,E2 -18212.29} C_VEL
LIN {X 0,Y 263.153,Z 338.7,A -85,B 0,C 180,E1 -18215.984,E2 -18215.984} C_VEL
LIN {X 0,Y 263.088,Z 338.67,A -85,B 0,C 180,E1 -18219.876,E2 -18219.876} C_VEL
LIN {X 0,Y 263.074,Z 338.714,A -85,B 0,C 180,E1 -18223.995,E2 -18223.995} C_VEL
LIN {X 0,Y 263.078,Z 338.694,A -85,B 0,C 180,E1 -18228.418,E2 -18228.418} C_VEL
LIN {X 0,Y 263.138,Z 338.685,A -85,B 0,C 180,E1 -18232.1,E2 -18232.1} C_VEL
LIN {X 0,Y 263.151,Z 338.7,A -85,B 0,C 180,E1 -18235.886,E2 -18235.886} C_VEL
LIN {X 0,Y 263.164,Z 338.896,A -85,B 0,C 180,E1 -18239.12,E2 -18239.12} C_VEL
LIN {X 0,Y 263.366,Z 339.782,A -85,B 0,C 180,E1 -18239.366,E2 -18239.366} C_VEL
LIN {X 0,Y 273.044,Z 357.944,A -85,B 0,C 180,E1 -18241.176,E2 -18241.176} C_VEL
LIN {X 0,Y 280.077,Z 373.068,A -85,B 0,C 180,E1 -18242.431,E2 -18242.431} C_VEL
LIN {X 0,Y 279.183,Z 418.195,A -85,B 0,C 180,E1 -18243.627,E2 -18243.627} C_VEL
LIN {X 0,Y 278.793,Z 431.732,A -85,B 0,C 180,E1 -18244.197,E2 -18244.197} C_VEL
LIN {X 0,Y 278.102,Z 443.513,A -85,B 0,C 180,E1 -18244.958,E2 -18244.958} C_VEL
LIN {X 0,Y 276.952,Z 455.754,A -85,B 0,C 180,E1 -18246.045,E2 -18246.045} C_VEL
LIN {X 0,Y 275.636,Z 466.021,A -85,B 0,C 180,E1 -18247.217,E2 -18247.217} C_VEL
LIN {X 0,Y 273.894,Z 476.765,A -85,B 0,C 180,E1 -18248.75,E2 -18248.75} C_VEL
LIN {X 0,Y 272.27,Z 485.958,A -85,B 0,C 180,E1 -18250.394,E2 -18250.394} C_VEL
LIN {X 0,Y 270.736,Z 494.307,A -85,B 0,C 180,E1 -18252.241,E2 -18252.241} C_VEL
LIN {X 0,Y 268.963,Z 502.423,A -85,B 0,C 180,E1 -18254.465,E2 -18254.465} C_VEL
LIN {X 0,Y 267.303,Z 509.53,A -85,B 0,C 180,E1 -18256.928,E2 -18256.928} C_VEL
LIN {X 0,Y 266.14,Z 514.903,A -85,B 0,C 180,E1 -18259.348,E2 -18259.348} C_VEL
LIN {X 0,Y 265.039,Z 518.793,A -85,B 0,C 180,E1 -18261.614,E2 -18261.614} C_VEL
LIN {X 0,Y 264.168,Z 521.669,A -85,B 0,C 180,E1 -18263.891,E2 -18263.891} C_VEL
LIN {X 0,Y 264.022,Z 523.008,A -85,B 0,C 180,E1 -18265.42,E2 -18265.42} C_VEL
LIN {X 0,Y 263.738,Z 523.984,A -85,B 0,C 180,E1 -18266.945,E2 -18266.945} C_VEL
LIN {X 0,Y 263.73,Z 524.562,A -85,B 0,C 180,E1 -18268.473,E2 -18268.473} C_VEL
LIN {X 0,Y 263.691,Z 524.786,A -85,B 0,C 180,E1 -18270,E2 -18270} C_VEL
LIN {X 0,Y 263.729,Z 524.599,A -85,B 0,C 180,E1 -18271.527,E2 -18271.527} C_VEL
LIN {X 0,Y 263.737,Z 524.044,A -85,B 0,C 180,E1 -18273.055,E2 -18273.055} C_VEL
LIN {X 0,Y 264.016,Z 523.092,A -85,B 0,C 180,E1 -18274.58,E2 -18274.58} C_VEL
LIN {X 0,Y 264.154,Z 521.793,A -85,B 0,C 180,E1 -18276.109,E2 -18276.109} C_VEL
LIN {X 0,Y 265.032,Z 518.962,A -85,B 0,C 180,E1 -18278.386,E2 -18278.386} C_VEL
LIN {X 0,Y 266.115,Z 515.131,A -85,B 0,C 180,E1 -18280.653,E2 -18280.653} C_VEL
LIN {X 0,Y 267.219,Z 510.048,A -85,B 0,C 180,E1 -18282.994,E2 -18282.994} C_VEL
LIN {X 0,Y 268.974,Z 502.802,A -85,B 0,C 180,E1 -18285.534,E2 -18285.534} C_VEL
LIN {X 0,Y 270.723,Z 494.771,A -85,B 0,C 180,E1 -18287.76,E2 -18287.76} C_VEL
LIN {X 0,Y 272.272,Z 486.544,A -85,B 0,C 180,E1 -18289.606,E2 -18289.606} C_VEL
LIN {X 0,Y 273.834,Z 477.502,A -85,B 0,C 180,E1 -18291.255,E2 -18291.255} C_VEL
LIN {X 0,Y 275.812,Z 465.952,A -85,B 0,C 180,E1 -18292.901,E2 -18292.901} C_VEL
LIN {X 0,Y 277.262,Z 454.014,A -85,B 0,C 180,E1 -18294.248,E2 -18294.248} C_VEL
LIN {X 0,Y 278.443,Z 441.407,A -85,B 0,C 180,E1 -18295.299,E2 -18295.299} C_VEL
LIN {X 0,Y 279.084,Z 428.97,A -85,B 0,C 180,E1 -18296.053,E2 -18296.053} C_VEL
LIN {X 0,Y 279.205,Z 418.87,A -85,B 0,C 180,E1 -18296.474,E2 -18296.474} C_VEL
LIN {X 0,Y 280.067,Z 378.422,A -85,B 0,C 180,E1 -18297.545,E2 -18297.545} C_VEL
LIN {X 0,Y 280.141,Z 373.204,A -85,B 0,C 180,E1 -18297.686,E2 -18297.686} C_VEL
LIN {X 0,Y 272.857,Z 357.475,A -85,B 0,C 180,E1 -18298.991,E2 -18298.991} C_VEL
LIN {X 0,Y 264.448,Z 341.992,A -85,B 0,C 180,E1 -18300.528,E2 -18300.528} C_VEL
LIN {X 0,Y 263.265,Z 339.39,A -85,B 0,C 180,E1 -18300.837,E2 -18300.837} C_VEL
LIN {X 0,Y 263.15,Z 338.743,A -85,B 0,C 180,E1 -18301.162,E2 -18301.162} C_VEL
LIN {X 0,Y 263.151,Z 338.699,A -85,B 0,C 180,E1 -18304.114,E2 -18304.114} C_VEL
LIN {X 0,Y 263.102,Z 338.689,A -85,B 0,C 180,E1 -18307.906,E2 -18307.906} C_VEL
LIN {X 0,Y 263.072,Z 338.692,A -85,B 0,C 180,E1 -18311.902,E2 -18311.902} C_VEL
LIN {X 0,Y 263.076,Z 338.714,A -85,B 0,C 180,E1 -18316.161,E2 -18316.161} C_VEL
LIN {X 0,Y 263.11,Z 338.666,A -85,B 0,C 180,E1 -18320.77,E2 -18320.77} C_VEL
LIN {X 0,Y 263.153,Z 338.699,A -85,B 0,C 180,E1 -18324.016,E2 -18324.016} C_VEL
LIN {X 0,Y 263.123,Z 338.682,A -85,B 0,C 180,E1 -18327.71,E2 -18327.71} C_VEL
LIN {X 0,Y 263.132,Z 338.655,A -85,B 0,C 180,E1 -18331.809,E2 -18331.809} C_VEL
LIN {X 0,Y 263.111,Z 338.712,A -85,B 0,C 180,E1 -18336.38,E2 -18336.38} C_VEL
LIN {X 0,Y 263.204,Z 338.683,A -85,B 0,C 180,E1 -18339.688,E2 -18339.688} C_VEL
LIN {X 0,Y 263.306,Z 338.668,A -85,B 0,C 180,E1 -18344.519,E2 -18344.519} C_VEL
LIN {X 0,Y 263.344,Z 338.68,A -85,B 0,C 180,E1 -18349.233,E2 -18349.233} C_VEL
LIN {X 0,Y 263.52,Z 338.639,A -85,B 0,C 180,E1 -18352.337,E2 -18352.337} C_VEL
LIN {X 0,Y 263.729,Z 338.613,A -85,B 0,C 180,E1 -18358.473,E2 -18358.473} C_VEL
LIN {X 0,Y 263.659,Z 338.636,A -85,B 0,C 180,E1 -18361.911,E2 -18361.911} C_VEL
LIN {X 0,Y 262.837,Z 338.744,A -85,B 0,C 180,E1 -18363.184,E2 -18363.184} C_VEL
LIN {X 0,Y 259.918,Z 339.095,A -85,B 0,C 180,E1 -18365.261,E2 -18365.261} C_VEL
LIN {X 0,Y 257.529,Z 339.392,A -85,B 0,C 180,E1 -18366.95,E2 -18366.95} C_VEL
LIN {X 0,Y 256.51,Z 339.526,A -85,B 0,C 180,E1 -18368.259,E2 -18368.259} C_VEL
LIN {X 0,Y 256.424,Z 339.535,A -85,B 0,C 180,E1 -18368.703,E2 -18368.703} C_VEL
LIN {X 0,Y 256.253,Z 339.544,A -85,B 0,C 180,E1 -18372.674,E2 -18372.674} C_VEL
LIN {X 0,Y 256.239,Z 339.568,A -85,B 0,C 180,E1 -18376.271,E2 -18376.271} C_VEL
LIN {X 0,Y 256.135,Z 339.541,A -85,B 0,C 180,E1 -18381.109,E2 -18381.109} C_VEL
LIN {X 0,Y 256.101,Z 339.583,A -85,B 0,C 180,E1 -18385.099,E2 -18385.099} C_VEL
LIN {X 0,Y 256.086,Z 339.558,A -85,B 0,C 180,E1 -18388.575,E2 -18388.575} C_VEL
LIN {X 0,Y 256.071,Z 339.589,A -85,B 0,C 180,E1 -18391.702,E2 -18391.702} C_VEL
LIN {X 0,Y 256.075,Z 339.569,A -85,B 0,C 180,E1 -18395.194,E2 -18395.194} C_VEL
LIN {X 0,Y 256.062,Z 339.574,A -85,B 0,C 180,E1 -18399.144,E2 -18399.144} C_VEL
LIN {X 0,Y 256.025,Z 339.561,A -85,B 0,C 180,E1 -18403.335,E2 -18403.335} C_VEL
LIN {X 0,Y 256.062,Z 339.785,A -85,B 0,C 180,E1 -18406.035,E2 -18406.035} C_VEL
LIN {X 0,Y 259.22,Z 351.028,A -85,B 0,C 180,E1 -18409.989,E2 -18409.989} C_VEL
LIN {X 0,Y 261.934,Z 362.218,A -85,B 0,C 180,E1 -18413.604,E2 -18413.604} C_VEL
LIN {X 0,Y 264.253,Z 373.318,A -85,B 0,C 180,E1 -18416.961,E2 -18416.961} C_VEL
LIN {X 0,Y 264.375,Z 374.985,A -85,B 0,C 180,E1 -18417.432,E2 -18417.432} C_VEL
LIN {X 0,Y 263.535,Z 379.77,A -85,B 0,C 180,E1 -18418.582,E2 -18418.582} C_VEL
LIN {X 0,Y 266.963,Z 405.486,A -85,B 0,C 180,E1 -18419.825,E2 -18419.825} C_VEL
LIN {X 0,Y 270.062,Z 434.645,A -85,B 0,C 180,E1 -18421.056,E2 -18421.056} C_VEL
LIN {X 0,Y 271.53,Z 454.188,A -85,B 0,C 180,E1 -18421.791,E2 -18421.791} C_VEL
LIN {X 0,Y 270.295,Z 491.957,A -85,B 0,C 180,E1 -18422.816,E2 -18422.816} C_VEL
LIN {X 0,Y 269.158,Z 505.593,A -85,B 0,C 180,E1 -18423.475,E2 -18423.475} C_VEL
LIN {X 0,Y 267.625,Z 517.577,A -85,B 0,C 180,E1 -18424.323,E2 -18424.323} C_VEL
LIN {X 0,Y 265.903,Z 528.762,A -85,B 0,C 180,E1 -18425.4,E2 -18425.4} C_VEL
LIN {X 0,Y 263.617,Z 540.41,A -85,B 0,C 180,E1 -18426.845,E2 -18426.845} C_VEL
LIN {X 0,Y 261.437,Z 550.943,A -85,B 0,C 180,E1 -18428.515,E2 -18428.515} C_VEL
LIN {X 0,Y 259.566,Z 559.587,A -85,B 0,C 180,E1 -18430.218,E2 -18430.218} C_VEL
LIN {X 0,Y 257.968,Z 567.618,A -85,B 0,C 180,E1 -18432.152,E2 -18432.152} C_VEL
LIN {X 0,Y 256.584,Z 574.293,A -85,B 0,C 180,E1 -18434.103,E2 -18434.103} C_VEL
LIN {X 0,Y 255.574,Z 580.938,A -85,B 0,C 180,E1 -18436.483,E2 -18436.483} C_VEL
LIN {X 0,Y 254.948,Z 586.252,A -85,B 0,C 180,E1 -18438.874,E2 -18438.874} C_VEL
LIN {X 0,Y 254.811,Z 590.433,A -85,B 0,C 180,E1 -18441.275,E2 -18441.275} C_VEL
LIN {X 0,Y 255.022,Z 593.568,A -85,B 0,C 180,E1 -18443.671,E2 -18443.671} C_VEL
LIN {X 0,Y 255.309,Z 595.086,A -85,B 0,C 180,E1 -18445.263,E2 -18445.263} C_VEL
LIN {X 0,Y 255.554,Z 596.175,A -85,B 0,C 180,E1 -18446.847,E2 -18446.847} C_VEL
LIN {X 0,Y 255.866,Z 596.861,A -85,B 0,C 180,E1 -18448.426,E2 -18448.426} C_VEL
LIN {X 0,Y 256.278,Z 597.142,A -85,B 0,C 180,E1 -18450,E2 -18450} C_VEL
LIN {X 0,Y 255.871,Z 596.852,A -85,B 0,C 180,E1 -18451.574,E2 -18451.574} C_VEL
LIN {X 0,Y 255.565,Z 596.163,A -85,B 0,C 180,E1 -18453.153,E2 -18453.153} C_VEL
LIN {X 0,Y 255.33,Z 595.07,A -85,B 0,C 180,E1 -18454.737,E2 -18454.737} C_VEL
LIN {X 0,Y 254.964,Z 592.615,A -85,B 0,C 180,E1 -18457.101,E2 -18457.101} C_VEL
LIN {X 0,Y 254.824,Z 589.089,A -85,B 0,C 180,E1 -18459.525,E2 -18459.525} C_VEL
LIN {X 0,Y 255.096,Z 584.522,A -85,B 0,C 180,E1 -18461.925,E2 -18461.925} C_VEL
LIN {X 0,Y 255.829,Z 578.77,A -85,B 0,C 180,E1 -18464.314,E2 -18464.314} C_VEL
LIN {X 0,Y 257.141,Z 571.089,A -85,B 0,C 180,E1 -18466.85,E2 -18466.85} C_VEL
LIN {X 0,Y 258.827,Z 562.813,A -85,B 0,C 180,E1 -18469.016,E2 -18469.016} C_VEL
LIN {X 0,Y 260.76,Z 553.809,A -85,B 0,C 180,E1 -18470.923,E2 -18470.923} C_VEL
LIN {X 0,Y 263.147,Z 542.784,A -85,B 0,C 180,E1 -18472.784,E2 -18472.784} C_VEL
LIN {X 0,Y 265.278,Z 531.667,A -85,B 0,C 180,E1 -18474.245,E2 -18474.245} C_VEL
LIN {X 0,Y 267.38,Z 519.248,A -85,B 0,C 180,E1 -18475.493,E2 -18475.493} C_VEL
LIN {X 0,Y 269.015,Z 506.341,A -85,B 0,C 180,E1 -18476.451,E2 -18476.451} C_VEL
LIN {X 0,Y 270.113,Z 493.497,A -85,B 0,C 180,E1 -18477.095,E2 -18477.095} C_VEL
LIN {X 0,Y 270.865,Z 474.85,A -85,B 0,C 180,E1 -18477.642,E2 -18477.642} C_VEL
LIN {X 0,Y 271.419,Z 452.496,A -85,B 0,C 180,E1 -18478.232,E2 -18478.232} C_VEL
LIN {X 0,Y 268.807,Z 422.677,A -85,B 0,C 180,E1 -18479.403,E2 -18479.403} C_VEL
LIN {X 0,Y 265.67,Z 395.698,A -85,B 0,C 180,E1 -18480.587,E2 -18480.587} C_VEL
LIN {X 0,Y 263.511,Z 379.52,A -85,B 0,C 180,E1 -18481.41,E2 -18481.41} C_VEL
LIN {X 0,Y 264.328,Z 374.841,A -85,B 0,C 180,E1 -18482.575,E2 -18482.575} C_VEL
LIN {X 0,Y 263.444,Z 369.229,A -85,B 0,C 180,E1 -18484.208,E2 -18484.208} C_VEL
LIN {X 0,Y 261.127,Z 358.74,A -85,B 0,C 180,E1 -18487.444,E2 -18487.444} C_VEL
LIN {X 0,Y 258.268,Z 347.551,A -85,B 0,C 180,E1 -18491.144,E2 -18491.144} C_VEL
LIN {X 0,Y 256.05,Z 339.682,A -85,B 0,C 180,E1 -18493.994,E2 -18493.994} C_VEL
LIN {X 0,Y 256.052,Z 339.585,A -85,B 0,C 180,E1 -18497.823,E2 -18497.823} C_VEL
LIN {X 0,Y 256.113,Z 339.506,A -85,B 0,C 180,E1 -18502.729,E2 -18502.729} C_VEL
LIN {X 0,Y 256.063,Z 339.574,A -85,B 0,C 180,E1 -18506.706,E2 -18506.706} C_VEL
LIN {X 0,Y 256.05,Z 339.568,A -85,B 0,C 180,E1 -18510.392,E2 -18510.392} C_VEL
LIN {X 0,Y 256.075,Z 339.581,A -85,B 0,C 180,E1 -18513.952,E2 -18513.952} C_VEL
